KUKA KRL program: MyProgram_259().src

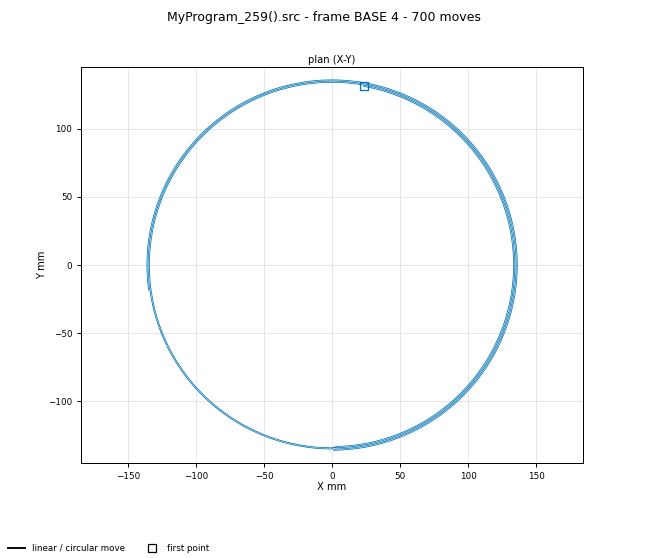
[picture p0: tool path of MyProgram_259().src in frame BASE 4, 700 of 700 moves have a stored position in this frame; points joined in program order, loops and branches not executed]
&ACCESS RVP
&REL 1
&PARAM TEMPLATE = C:\KRC\Roboter\Template\vorgabe
&PARAM EDITMASK = *
DEF MyProgram_259()
; ---- Setting reference (Base) ----
$BASE = BASE_DATA[4]

; --------------------------
; ---- Setting tool (TCP) ----
$TOOL = TOOL_DATA[3]
; --------------------------

$VEL.CP = VEL_APROX_PRINT
Startdeposition()
$VEL.CP = VEL_PRINT
LIN {X 23.111,Y 131.2816,Z 167,A 79.654,B 11.3384,C -0.0148,E1 11.3678,E2 371.0348} C_DIS
LIN {X 26.5577,Y 130.6274,Z 167,A 78.0949,B 11.3384,C -0.0129,E1 11.3721,E2 372.5994} C_DIS
LIN {X 29.5661,Y 129.9795,Z 167,A 76.8546,B 11.3384,C -0.0141,E1 11.3755,E2 373.8297} C_DIS
LIN {X 32.4376,Y 129.2932,Z 167,A 75.5169,B 11.3384,C -0.0116,E1 11.3791,E2 375.1753} C_DIS
LIN {X 34.9908,Y 128.6268,Z 167,A 73.9813,B 11.3384,C -0.0011,E1 11.3834,E2 376.758} C_DIS
LIN {X 38.5081,Y 127.6173,Z 167,A 72.9209,B 11.3384,C -0.0122,E1 11.3861,E2 377.7578} C_DIS
LIN {X 42.8444,Y 126.2288,Z 167,A 70.7155,B 11.3384,C -0.0045,E1 11.392,E2 379.9924} C_DIS
LIN {X 46.2522,Y 125.0191,Z 167,A 69.2886,B 11.3384,C -0.0061,E1 11.3957,E2 381.4041} C_DIS
LIN {X 50.6858,Y 123.2893,Z 167,A 67.2139,B 11.3384,C -0.0033,E1 11.4011,E2 383.4822} C_DIS
LIN {X 54.1145,Y 121.8215,Z 167,A 65.658,B 11.3384,C -0.0027,E1 11.4051,E2 385.0325} C_DIS
LIN {X 57.2968,Y 120.3572,Z 167,A 64.0803,B 11.3384,C 0.0009,E1 11.4091,E2 386.6187} C_DIS
LIN {X 61.2926,Y 118.3745,Z 167,A 62.2048,B 11.3384,C 0.0023,E1 11.4137,E2 388.4895} C_DIS
LIN {X 64.6789,Y 116.5587,Z 167,A 60.1894,B 11.3384,C 0.0136,E1 11.4188,E2 390.5479} C_DIS
LIN {X 68.1241,Y 114.5792,Z 167,A 58.8253,B 11.3384,C 0.0075,E1 11.422,E2 391.8717} C_DIS
LIN {X 71.9938,Y 112.1881,Z 167,A 56.8981,B 11.3384,C 0.0098,E1 11.4265,E2 393.7959} C_DIS
LIN {X 77.218,Y 108.6591,Z 167,A 54.1798,B 11.3384,C 0.0144,E1 11.4328,E2 396.5158} C_DIS
LIN {X 80.7271,Y 106.0778,Z 167,A 51.9721,B 11.3384,C 0.026,E1 11.4378,E2 398.7636} C_DIS
LIN {X 83.987,Y 103.5161,Z 167,A 50.5474,B 11.3384,C 0.0203,E1 11.4408,E2 400.1466} C_DIS
LIN {X 87.3612,Y 100.6848,Z 167,A 48.6571,B 11.3384,C 0.0237,E1 11.4448,E2 402.0372} C_DIS
LIN {X 90.7212,Y 97.6676,Z 167,A 46.7628,B 11.3384,C 0.0263,E1 11.4487,E2 403.9266} C_DIS
LIN {X 93.9495,Y 94.5662,Z 167,A 44.8876,B 11.3384,C 0.0289,E1 11.4524,E2 405.7967} C_DIS
LIN {X 97.0915,Y 91.3375,Z 167,A 42.9827,B 11.3384,C 0.0321,E1 11.4561,E2 407.6987} C_DIS
LIN {X 100.0588,Y 88.0771,Z 167,A 41.1296,B 11.3384,C 0.0351,E1 11.4596,E2 409.5477} C_DIS
LIN {X 102.7672,Y 84.9011,Z 167,A 38.5566,B 11.3384,C 0.0591,E1 11.4643,E2 412.2138} C_DIS
LIN {X 106.531,Y 80.1277,Z 167,A 36.9658,B 11.3384,C 0.0388,E1 11.4668,E2 413.6849} C_DIS
LIN {X 109.5214,Y 75.9892,Z 167,A 34.5744,B 11.3384,C 0.0491,E1 11.4707,E2 416.1011} C_DIS
LIN {X 111.9973,Y 72.291,Z 167,A 32.6754,B 11.3384,C 0.0533,E1 11.4737,E2 417.9997} C_DIS
LIN {X 113.8063,Y 69.4083,Z 167,A 30.2613,B 11.3382,C 0.0816,E1 11.4773,E2 420.5274} C_DIS
LIN {X 117.3478,Y 63.2361,Z 167,A 28.3,B 11.3383,C 0.0609,E1 11.4798,E2 422.3608} C_DIS
LIN {X 120.1649,Y 57.6993,Z 167,A 25.6079,B 11.3383,C 0.0684,E1 11.4832,E2 425.0575} C_DIS
LIN {X 121.4581,Y 54.9269,Z 167,A 24.248,B 11.3383,C 0.0731,E1 11.4847,E2 426.4238} C_DIS
LIN {X 122.6861,Y 52.1301,Z 167,A 22.924,B 11.3383,C 0.0769,E1 11.4862,E2 427.7503} C_DIS
LIN {X 124.6025,Y 47.3646,Z 167,A 20.8006,B 11.3382,C 0.0806,E1 11.4884,E2 429.8652} C_DIS
LIN {X 125.7921,Y 44.1059,Z 167,A 19.5229,B 11.3382,C 0.0791,E1 11.4896,E2 431.1185} C_DIS
LIN {X 127.1799,Y 39.931,Z 167,A 17.2589,B 11.3381,C 0.0942,E1 11.4915,E2 433.429} C_DIS
LIN {X 128.6725,Y 34.8197,Z 167,A 15.1937,B 11.3381,C 0.0947,E1 11.4931,E2 435.4693} C_DIS
LIN {X 129.5781,Y 31.2779,Z 167,A 13.6311,B 11.3381,C 0.0989,E1 11.4941,E2 437.0322} C_DIS
LIN {X 130.56,Y 26.8888,Z 167,A 11.7393,B 11.3381,C 0.1034,E1 11.4953,E2 438.9209} C_DIS
LIN {X 131.2572,Y 23.2472,Z 167,A 10.156,B 11.338,C 0.1077,E1 11.4961,E2 440.5045} C_DIS
LIN {X 131.9587,Y 18.8608,Z 167,A 8.3069,B 11.338,C 0.1116,E1 11.4968,E2 442.3481} C_DIS
LIN {X 132.4922,Y 14.6572,Z 167,A 6.5104,B 11.3379,C 0.1163,E1 11.4974,E2 444.1434} C_DIS
LIN {X 132.8356,Y 11.1164,Z 167,A 5.002,B 11.3379,C 0.1202,E1 11.4978,E2 445.6509} C_DIS
LIN {X 133.1209,Y 6.9099,Z 167,A 3.2192,B 11.3379,C 0.1247,E1 11.4981,E2 447.432} C_DIS
LIN {X 133.2576,Y 3.3765,Z 167,A 1.6311,B 11.3377,C 0.131,E1 11.4983,E2 449.0299} C_DIS
LIN {X 133.2963,Y -1.0793,Z 167,A -0.2205,B 11.3377,C 0.135,E1 11.4983,E2 450.8758} C_DIS
LIN {X 133.166,Y -6.0129,Z 167,A -2.6544,B 11.3375,C 0.1496,E1 11.498,E2 453.3496} C_DIS
LIN {X 132.9435,Y -9.7408,Z 167,A -3.8408,B 11.3375,C 0.1431,E1 11.4978,E2 454.4872} C_DIS
LIN {X 132.5722,Y -13.9132,Z 167,A -5.6427,B 11.3375,C 0.1484,E1 11.4973,E2 456.2913} C_DIS
LIN {X 132.1367,Y -17.5729,Z 167,A -7.2609,B 11.3375,C 0.154,E1 11.4967,E2 457.9154} C_DIS
LIN {X 131.5062,Y -21.7936,Z 167,A -9.0238,B 11.3375,C 0.1574,E1 11.496,E2 459.6716} C_DIS
LIN {X 130.8011,Y -25.6973,Z 167,A -10.6485,B 11.3374,C 0.1603,E1 11.4951,E2 461.2886} C_DIS
LIN {X 130.0562,Y -29.2303,Z 167,A -12.2687,B 11.3373,C 0.1666,E1 11.4942,E2 462.9187} C_DIS
LIN {X 127.6873,Y -38.2794,Z 167,A -16.8884,B 11.3368,C 0.1941,E1 11.4907,E2 467.6153} C_DIS
LIN {X 126.0223,Y -43.4421,Z 167,A -18.4516,B 11.3371,C 0.1802,E1 11.4894,E2 469.0884} C_DIS
LIN {X 124.9261,Y -46.5005,Z 167,A -20.042,B 11.3369,C 0.1893,E1 11.4878,E2 470.704} C_DIS
LIN {X 123.1296,Y -51.0683,Z 167,A -21.9539,B 11.3369,C 0.1899,E1 11.4858,E2 472.5943} C_DIS
LIN {X 121.6299,Y -54.5429,Z 167,A -23.6333,B 11.3369,C 0.1957,E1 11.4839,E2 474.2819} C_DIS
LIN {X 118.9639,Y -60.137,Z 167,A -26.2388,B 11.3367,C 0.2014,E1 11.4808,E2 476.8835} C_DIS
LIN {X 117.2059,Y -63.4995,Z 167,A -27.7083,B 11.3367,C 0.2014,E1 11.4789,E2 478.3353} C_DIS
LIN {X 115.8849,Y -65.8787,Z 167,A -29.0352,B 11.3366,C 0.2087,E1 11.477,E2 479.6826} C_DIS
LIN {X 113.6486,Y -69.6653,Z 167,A -30.9028,B 11.3366,C 0.213,E1 11.4743,E2 481.5497} C_DIS
LIN {X 111.1338,Y -73.6117,Z 167,A -32.8818,B 11.3364,C 0.2172,E1 11.4713,E2 483.5271} C_DIS
LIN {X 108.6815,Y -77.1866,Z 167,A -34.7672,B 11.3364,C 0.2224,E1 11.4683,E2 485.4173} C_DIS
LIN {X 106.0494,Y -80.7643,Z 167,A -36.6339,B 11.3363,C 0.2259,E1 11.4652,E2 487.2809} C_DIS
LIN {X 103.5315,Y -83.968,Z 167,A -38.5461,B 11.3361,C 0.2343,E1 11.4618,E2 489.2146} C_DIS
LIN {X 99.5166,Y -88.6895,Z 167,A -41.0194,B 11.3361,C 0.2354,E1 11.4573,E2 491.6677} C_DIS
LIN {X 96.4218,Y -92.044,Z 167,A -43.0399,B 11.3359,C 0.2413,E1 11.4534,E2 493.6974} C_DIS
LIN {X 93.3721,Y -95.1363,Z 167,A -44.8374,B 11.3359,C 0.2436,E1 11.4499,E2 495.4886} C_DIS
LIN {X 89.6728,Y -98.631,Z 167,A -46.9436,B 11.3359,C 0.246,E1 11.4456,E2 497.5872} C_DIS
LIN {X 86.5709,Y -101.3649,Z 167,A -49.0209,B 11.3356,C 0.2574,E1 11.4411,E2 499.7029} C_DIS
LIN {X 83.6178,Y -103.8139,Z 167,A -50.5259,B 11.3356,C 0.2569,E1 11.4379,E2 501.1921} C_DIS
LIN {X 79.3097,Y -107.1419,Z 167,A -52.6562,B 11.3356,C 0.2559,E1 11.4332,E2 503.2993} C_DIS
LIN {X 76.0282,Y -109.4943,Z 167,A -54.1959,B 11.3356,C 0.254,E1 11.4297,E2 504.8168} C_DIS
LIN {X 71.2074,Y -112.6889,Z 167,A -56.8197,B 11.3355,C 0.2618,E1 11.4236,E2 507.4599} C_DIS
LIN {X 67.5869,Y -114.8968,Z 167,A -58.6507,B 11.3355,C 0.265,E1 11.4192,E2 509.2937} C_DIS
LIN {X 63.8199,Y -117.0312,Z 167,A -60.4111,B 11.3355,C 0.2653,E1 11.4149,E2 511.0435} C_DIS
LIN {X 60.7742,Y -118.6395,Z 167,A -61.7629,B 11.3355,C 0.2642,E1 11.4116,E2 512.3809} C_DIS
LIN {X 57.705,Y -120.1622,Z 167,A -63.3149,B 11.3353,C 0.2683,E1 11.4077,E2 513.9439} C_DIS
LIN {X 54.7635,Y -121.5313,Z 167,A -64.6557,B 11.3353,C 0.2688,E1 11.4043,E2 515.2793} C_DIS
LIN {X 50.7074,Y -123.2803,Z 167,A -66.7419,B 11.3352,C 0.2759,E1 11.3988,E2 517.3901} C_DIS
LIN {X 47.1663,Y -124.6768,Z 167,A -68.2475,B 11.3352,C 0.2746,E1 11.395,E2 518.8811} C_DIS
LIN {X 44.1745,Y -125.7683,Z 167,A -70.4197,B 11.3347,C 0.2961,E1 11.389,E2 521.1519} C_DIS
LIN {X 38.5187,Y -127.6141,Z 167,A -71.8598,B 11.3353,C 0.2709,E1 11.3855,E2 522.4583} C_DIS
LIN {X 32.3264,Y -129.3214,Z 167,A -75.0203,B 11.335,C 0.2834,E1 11.3769,E2 525.6698} C_DIS
LIN {X 28.9097,Y -130.1294,Z 167,A -76.5137,B 11.335,C 0.2842,E1 11.3728,E2 527.1625} C_DIS
LIN {X 25.3413,Y -130.8692,Z 167,A -78.0214,B 11.335,C 0.2838,E1 11.3687,E2 528.6639} C_DIS
LIN {X 21.8863,Y -131.4908,Z 167,A -79.4748,B 11.335,C 0.2834,E1 11.3647,E2 530.1116} C_DIS
LIN {X 18.2129,Y -132.0513,Z 167,A -81.1212,B 11.335,C 0.2855,E1 11.3601,E2 531.7651} C_DIS
LIN {X 14.4448,Y -132.515,Z 167,A -82.6877,B 11.335,C 0.2847,E1 11.3558,E2 533.3245} C_DIS
LIN {X 11.1181,Y -132.8355,Z 167,A -84.1509,B 11.335,C 0.2859,E1 11.3517,E2 534.7917} C_DIS
LIN {X 6.9099,Y -133.1209,Z 167,A -85.9699,B 11.335,C 0.2866,E1 11.3466,E2 536.6125} C_DIS
LIN {X 3.1394,Y -133.2642,Z 167,A -87.6442,B 11.3349,C 0.2883,E1 11.3419,E2 538.294} C_DIS
LIN {X 3.1394,Y -133.2642,Z 167,A -87.6442,B 11.3349,C 0.2883,E1 11.3419,E2 538.294} C_DIS
Enddeposition()
LIN {X 0.9649,Y -134.2111,Z 167,A -88.1707,B 11.0146,C 0.3002,E1 11.0204,E2 538.9013} C_DIS
Startdeposition()
$VEL.CP = VEL_PRINT
LIN {X 3.4581,Y -134.1713,Z 167,A -86.6173,B 11.0149,C 0.2884,E1 11.0249,E2 537.2868} C_DIS
LIN {X 7.1388,Y -134.0261,Z 167,A -85.0914,B 11.0149,C 0.2891,E1 11.0291,E2 535.7658} C_DIS
LIN {X 11.0919,Y -133.7565,Z 167,A -83.3861,B 11.0149,C 0.2882,E1 11.0339,E2 534.0579} C_DIS
LIN {X 14.5172,Y -133.4281,Z 167,A -81.9055,B 11.0149,C 0.2873,E1 11.038,E2 532.575} C_DIS
LIN {X 17.6741,Y -133.0468,Z 167,A -80.5898,B 11.0149,C 0.2876,E1 11.0416,E2 531.2637} C_DIS
LIN {X 20.9035,Y -132.5781,Z 167,A -79.2392,B 11.0149,C 0.2878,E1 11.0454,E2 529.9175} C_DIS
LIN {X 23.8519,Y -132.0791,Z 167,A -77.8862,B 11.015,C 0.2852,E1 11.0491,E2 528.5541} C_DIS
LIN {X 27.4798,Y -131.374,Z 167,A -76.2645,B 11.015,C 0.283,E1 11.0536,E2 526.926} C_DIS
LIN {X 31.1737,Y -130.5451,Z 167,A -74.6858,B 11.015,C 0.2826,E1 11.0578,E2 525.3507} C_DIS
LIN {X 37.1831,Y -128.9629,Z 167,A -72.1203,B 11.015,C 0.2824,E1 11.0647,E2 522.7943} C_DIS
LIN {X 41.6665,Y -127.5844,Z 167,A -69.7848,B 11.0153,C 0.2721,E1 11.0711,E2 520.4156} C_DIS
LIN {X 44.8752,Y -126.4926,Z 167,A -68.7096,B 11.0151,C 0.2798,E1 11.0738,E2 519.3857} C_DIS
LIN {X 47.7371,Y -125.4407,Z 167,A -67.2008,B 11.0153,C 0.2731,E1 11.0778,E2 517.8501} C_DIS
LIN {X 51.3045,Y -124.0231,Z 167,A -65.8734,B 11.0152,C 0.2789,E1 11.0811,E2 516.56} C_DIS
LIN {X 53.6246,Y -123.0375,Z 167,A -64.6565,B 11.0152,C 0.274,E1 11.0843,E2 515.3247} C_DIS
LIN {X 56.6,Y -121.6971,Z 167,A -63.2535,B 11.0153,C 0.2719,E1 11.0879,E2 513.9192} C_DIS
LIN {X 60.1418,Y -119.9889,Z 167,A -61.6059,B 11.0153,C 0.2703,E1 11.092,E2 512.274} C_DIS
LIN {X 63.0439,Y -118.489,Z 167,A -60.1857,B 11.0154,C 0.2676,E1 11.0955,E2 510.8494} C_DIS
LIN {X 66.5933,Y -116.5313,Z 167,A -58.4086,B 11.0155,C 0.2637,E1 11.0999,E2 509.0649} C_DIS
LIN {X 70.5341,Y -114.1898,Z 167,A -56.2378,B 11.0157,C 0.255,E1 11.1051,E2 506.8655} C_DIS
LIN {X 73.337,Y -112.4092,Z 167,A -54.7783,B 11.0158,C 0.2515,E1 11.1085,E2 505.3993} C_DIS
LIN {X 76.4215,Y -110.336,Z 167,A -53.5539,B 11.0157,C 0.258,E1 11.1113,E2 504.2187} C_DIS
LIN {X 79.6868,Y -108.0014,Z 167,A -51.5499,B 11.0159,C 0.2474,E1 11.1159,E2 502.1767} C_DIS
LIN {X 82.426,Y -105.9255,Z 167,A -50.5266,B 11.0157,C 0.2561,E1 11.118,E2 501.2073} C_DIS
LIN {X 87.7566,Y -101.553,Z 167,A -47.6665,B 11.0157,C 0.2525,E1 11.1242,E2 498.3548} C_DIS
LIN {X 92.6598,Y -97.0998,Z 167,A -44.6294,B 11.016,C 0.2412,E1 11.1305,E2 495.2887} C_DIS
LIN {X 95.2574,Y -94.5527,Z 167,A -42.9732,B 11.0162,C 0.2352,E1 11.1337,E2 493.618} C_DIS
LIN {X 98.363,Y -91.3179,Z 167,A -40.9009,B 11.0163,C 0.2268,E1 11.1377,E2 491.5238} C_DIS
LIN {X 100.8242,Y -88.5928,Z 167,A -39.0555,B 11.0166,C 0.2158,E1 11.1412,E2 489.6418} C_DIS
LIN {X 104.2283,Y -84.5624,Z 167,A -37.4959,B 11.0163,C 0.2288,E1 11.1438,E2 488.1666} C_DIS
LIN {X 106.7196,Y -81.395,Z 167,A -35.7052,B 11.0164,C 0.2228,E1 11.1469,E2 486.3652} C_DIS
LIN {X 109.3532,Y -77.8213,Z 167,A -33.8282,B 11.0165,C 0.2187,E1 11.15,E2 484.4882} C_DIS
LIN {X 111.8562,Y -74.1793,Z 167,A -31.9264,B 11.0166,C 0.2135,E1 11.1529,E2 482.5825} C_DIS
LIN {X 114.2768,Y -70.3923,Z 167,A -30.0485,B 11.0166,C 0.2097,E1 11.1557,E2 480.7075} C_DIS
LIN {X 116.627,Y -66.4255,Z 167,A -28.3583,B 11.0166,C 0.212,E1 11.1581,E2 479.0496} C_DIS
LIN {X 118.0933,Y -63.7829,Z 167,A -26.7976,B 11.0168,C 0.2014,E1 11.1602,E2 477.4538} C_DIS
LIN {X 120.0797,Y -59.9578,Z 167,A -25.1134,B 11.0168,C 0.2006,E1 11.1623,E2 475.7869} C_DIS
LIN {X 122.5989,Y -54.6188,Z 167,A -23.0142,B 11.0168,C 0.205,E1 11.1648,E2 473.737} C_DIS
LIN {X 123.5234,Y -52.5008,Z 167,A -21.5505,B 11.017,C 0.1896,E1 11.1664,E2 472.2131} C_DIS
LIN {X 125.265,Y -48.1931,Z 167,A -19.6114,B 11.0171,C 0.1853,E1 11.1684,E2 470.2773} C_DIS
LIN {X 126.4758,Y -44.922,Z 167,A -17.9558,B 11.0172,C 0.1767,E1 11.17,E2 468.5993} C_DIS
LIN {X 127.8925,Y -40.7091,Z 167,A -16.3587,B 11.0172,C 0.1793,E1 11.1713,E2 467.0373} C_DIS
LIN {X 128.9537,Y -37.2145,Z 167,A -13.9995,B 11.0176,C 0.1534,E1 11.1732,E2 464.5766} C_DIS
LIN {X 130.4933,Y -31.3885,Z 167,A -12.4345,B 11.0173,C 0.173,E1 11.1742,E2 463.1344} C_DIS
LIN {X 131.1608,Y -28.4709,Z 167,A -11.0132,B 11.0174,C 0.1655,E1 11.1751,E2 461.6939} C_DIS
LIN {X 131.8437,Y -25.1198,Z 167,A -9.5944,B 11.0174,C 0.1624,E1 11.1758,E2 460.2785} C_DIS
LIN {X 132.4581,Y -21.6521,Z 167,A -8.115,B 11.0175,C 0.1586,E1 11.1765,E2 458.8005} C_DIS
LIN {X 132.9732,Y -18.2335,Z 167,A -6.4935,B 11.0176,C 0.1504,E1 11.1772,E2 457.1594} C_DIS
LIN {X 133.447,Y -14.3415,Z 167,A -4.9675,B 11.0176,C 0.1495,E1 11.1777,E2 455.6498} C_DIS
LIN {X 133.8003,Y -10.5737,Z 167,A -3.0213,B 11.0178,C 0.1359,E1 11.1781,E2 453.6609} C_DIS
LIN {X 134.0321,Y -7.0191,Z 167,A -2.0944,B 11.0177,C 0.1473,E1 11.1783,E2 452.8058} C_DIS
LIN {X 134.1683,Y -3.5667,Z 167,A -0.4639,B 11.0177,C 0.1388,E1 11.1784,E2 451.1547} C_DIS
LIN {X 134.2162,Y 0.2718,Z 167,A 1.2538,B 11.0179,C 0.1319,E1 11.1784,E2 449.4255} C_DIS
LIN {X 134.1522,Y 4.1432,Z 167,A 2.7921,B 11.0179,C 0.1301,E1 11.1784,E2 447.8997} C_DIS
LIN {X 133.9748,Y 8.0368,Z 167,A 4.4428,B 11.0179,C 0.1255,E1 11.1781,E2 446.249} C_DIS
LIN {X 133.745,Y 11.2285,Z 167,A 5.8177,B 11.0179,C 0.1213,E1 11.1778,E2 444.8715} C_DIS
LIN {X 133.4295,Y 14.5046,Z 167,A 7.2042,B 11.018,C 0.1177,E1 11.1774,E2 443.486} C_DIS
LIN {X 132.9148,Y 18.6428,Z 167,A 9.0024,B 11.018,C 0.1121,E1 11.1767,E2 441.6838} C_DIS
LIN {X 132.352,Y 22.2878,Z 167,A 10.5432,B 11.0181,C 0.1084,E1 11.1761,E2 440.1457} C_DIS
LIN {X 131.5324,Y 26.7015,Z 167,A 12.4115,B 11.0181,C 0.1042,E1 11.1751,E2 438.2816} C_DIS
LIN {X 130.7762,Y 30.1897,Z 167,A 13.9008,B 11.0181,C 0.1008,E1 11.1742,E2 436.7951} C_DIS
LIN {X 129.774,Y 34.2426,Z 167,A 15.687,B 11.0182,C 0.0956,E1 11.1729,E2 435.0068} C_DIS
LIN {X 128.713,Y 38.0367,Z 167,A 17.8826,B 11.0184,C 0.0773,E1 11.1712,E2 432.7464} C_DIS
LIN {X 127.2912,Y 42.5521,Z 167,A 19.3912,B 11.0184,C 0.0853,E1 11.1699,E2 431.2993} C_DIS
LIN {X 125.6178,Y 47.2642,Z 167,A 21.5575,B 11.0184,C 0.0786,E1 11.1678,E2 429.1275} C_DIS
LIN {X 124.3162,Y 50.5902,Z 167,A 22.9402,B 11.0184,C 0.0782,E1 11.1664,E2 427.761} C_DIS
LIN {X 123.0436,Y 53.6106,Z 167,A 24.3908,B 11.0184,C 0.0731,E1 11.1648,E2 426.303} C_DIS
LIN {X 121.2172,Y 57.6205,Z 167,A 26.6027,B 11.0184,C 0.0595,E1 11.1621,E2 424.0491} C_DIS
LIN {X 119.4032,Y 61.2922,Z 167,A 27.8665,B 11.0184,C 0.0677,E1 11.1606,E2 422.8436} C_DIS
LIN {X 117.7875,Y 64.3453,Z 167,A 30.052,B 11.0186,C 0.0453,E1 11.1575,E2 420.5697} C_DIS
LIN {X 115.0538,Y 69.1157,Z 167,A 31.6805,B 11.0185,C 0.0583,E1 11.1553,E2 419.0281} C_DIS
LIN {X 112.9618,Y 72.4834,Z 167,A 33.4274,B 11.0185,C 0.0527,E1 11.1527,E2 417.2735} C_DIS
LIN {X 110.5086,Y 76.1717,Z 167,A 35.5581,B 11.0185,C 0.0419,E1 11.1493,E2 415.1123} C_DIS
LIN {X 108.4311,Y 79.1016,Z 167,A 36.8459,B 11.0185,C 0.0447,E1 11.1473,E2 413.8538} C_DIS
LIN {X 104.0946,Y 84.7265,Z 167,A 39.6481,B 11.0185,C 0.0438,E1 11.1425,E2 411.078} C_DIS
LIN {X 101.8923,Y 87.3627,Z 167,A 41.2888,B 11.0185,C 0.0361,E1 11.1395,E2 409.4154} C_DIS
LIN {X 98.9133,Y 90.7214,Z 167,A 43.137,B 11.0185,C 0.0337,E1 11.136,E2 407.5747} C_DIS
LIN {X 96.0763,Y 93.7212,Z 167,A 44.944,B 11.0186,C 0.0289,E1 11.1325,E2 405.7616} C_DIS
LIN {X 92.8275,Y 96.9395,Z 167,A 46.8552,B 11.0186,C 0.026,E1 11.1287,E2 403.8546} C_DIS
LIN {X 89.4146,Y 100.0962,Z 167,A 48.8088,B 11.0186,C 0.023,E1 11.1247,E2 401.9041} C_DIS
LIN {X 85.9783,Y 103.0635,Z 167,A 50.7296,B 11.0186,C 0.0198,E1 11.1206,E2 399.9848} C_DIS
LIN {X 80.098,Y 107.6964,Z 167,A 54.5537,B 11.0186,C -0.0016,E1 11.1119,E2 396.0832} C_DIS
LIN {X 75.4981,Y 110.97,Z 167,A 56.1084,B 11.0186,C 0.016,E1 11.1086,E2 394.6322} C_DIS
LIN {X 72.82,Y 112.7455,Z 167,A 57.6162,B 11.0186,C 0.0104,E1 11.105,E2 393.1078} C_DIS
LIN {X 69.1453,Y 115.0359,Z 167,A 59.8176,B 11.0186,C -0.0011,E1 11.0997,E2 390.8633} C_DIS
LIN {X 65.8028,Y 116.9795,Z 167,A 61.1132,B 11.0186,C 0.0054,E1 11.0966,E2 389.6106} C_DIS
LIN {X 62.0142,Y 119.0297,Z 167,A 62.8825,B 11.0186,C 0.0047,E1 11.0923,E2 387.8495} C_DIS
LIN {X 59.3391,Y 120.385,Z 167,A 64.1738,B 11.0186,C 0.0028,E1 11.0891,E2 386.5568} C_DIS
LIN {X 56.0192,Y 121.9657,Z 167,A 65.6933,B 11.0186,C 0.0021,E1 11.0852,E2 385.0434} C_DIS
LIN {X 52.8538,Y 123.3708,Z 167,A 67.2391,B 11.0186,C -0.0012,E1 11.0813,E2 383.4895} C_DIS
LIN {X 48.4852,Y 125.1515,Z 167,A 69.1967,B 11.0186,C -0.0019,E1 11.0762,E2 381.5388} C_DIS
LIN {X 44.9095,Y 126.4802,Z 167,A 70.7713,B 11.0186,C -0.0021,E1 11.0721,E2 379.9709} C_DIS
LIN {X 41.0761,Y 127.7753,Z 167,A 72.4779,B 11.0186,C -0.0032,E1 11.0676,E2 378.2669} C_DIS
LIN {X 36.346,Y 129.2003,Z 167,A 74.3767,B 11.0186,C 0.0002,E1 11.0626,E2 376.3937} C_DIS
LIN {X 33.4824,Y 129.9726,Z 167,A 75.9585,B 11.0186,C -0.0082,E1 11.0582,E2 374.7742} C_DIS
LIN {X 29.8794,Y 130.8471,Z 167,A 77.4687,B 11.0186,C -0.0075,E1 11.0541,E2 373.2731} C_DIS
LIN {X 26.6862,Y 131.5355,Z 167,A 78.8545,B 11.0186,C -0.008,E1 11.0503,E2 371.8887} C_DIS
LIN {X 23.5582,Y 132.1316,Z 167,A 80.2365,B 11.0186,C -0.0092,E1 11.0465,E2 370.5043} C_DIS
LIN {X 19.7626,Y 132.7547,Z 167,A 81.8258,B 11.0186,C -0.0086,E1 11.0421,E2 368.9219} C_DIS
LIN {X 16.2843,Y 133.2244,Z 167,A 83.4219,B 11.0186,C -0.0114,E1 11.0377,E2 367.3145} C_DIS
LIN {X 12.6554,Y 133.6176,Z 167,A 84.9258,B 11.0186,C -0.0105,E1 11.0335,E2 365.8177} C_DIS
LIN {X 8.378,Y 133.9538,Z 167,A 86.7607,B 11.0186,C -0.0109,E1 11.0284,E2 363.9831} C_DIS
LIN {X 4.659,Y 134.1359,Z 167,A 88.3908,B 11.0186,C -0.0119,E1 11.0239,E2 362.3488} C_DIS
LIN {X 0.7067,Y 134.2137,Z 167,A 90.0012,B 11.0186,C -0.0102,E1 11.0194,E2 360.7485} C_DIS
LIN {X -3.1537,Y 134.1797,Z 167,A 91.7456,B 11.0186,C -0.0122,E1 11.0145,E2 358.9933} C_DIS
LIN {X -7.024,Y 134.0319,Z 167,A 93.4354,B 11.0186,C -0.0127,E1 11.0098,E2 357.2999} C_DIS
LIN {X -11.2551,Y 133.7427,Z 167,A 95.1269,B 11.0186,C -0.0095,E1 11.0051,E2 355.6237} C_DIS
LIN {X -14.8408,Y 133.3933,Z 167,A 96.6516,B 11.0186,C -0.0087,E1 11.0009,E2 354.1015} C_DIS
LIN {X -18.5922,Y 132.922,Z 167,A 98.3458,B 11.0186,C -0.0098,E1 10.9962,E2 352.3986} C_DIS
LIN {X -22.3311,Y 132.3448,Z 167,A 99.9063,B 11.0186,C -0.0077,E1 10.9919,E2 350.8456} C_DIS
LIN {X -26.2813,Y 131.6179,Z 167,A 102.4045,B 11.0186,C -0.0243,E1 10.9848,E2 348.254} C_DIS
LIN {X -31.9508,Y 130.3577,Z 167,A 103.8647,B 11.0186,C 0.0003,E1 10.9812,E2 346.9183} C_DIS
LIN {X -37.324,Y 128.9217,Z 167,A 107.0422,B 11.0186,C -0.0156,E1 10.9723,E2 343.6461} C_DIS
LIN {X -41.7584,Y 127.5555,Z 167,A 108.6732,B 11.0186,C -0.0059,E1 10.9681,E2 342.0589} C_DIS
LIN {X -45.7248,Y 126.1863,Z 167,A 110.2459,B 11.0186,C 0.0007,E1 10.9641,E2 340.5137} C_DIS
LIN {X -48.5561,Y 125.1239,Z 167,A 111.5711,B 11.0186,C 0.0014,E1 10.9606,E2 339.1854} C_DIS
LIN {X -51.5415,Y 123.9241,Z 167,A 113.1191,B 11.0186,C -0.0008,E1 10.9565,E2 337.6176} C_DIS
LIN {X -55.4809,Y 122.2133,Z 167,A 114.8021,B 11.0186,C 0.0047,E1 10.9523,E2 335.9543} C_DIS
LIN {X -58.4461,Y 120.8228,Z 167,A 116.1979,B 11.0186,C 0.0066,E1 10.9488,E2 334.5599} C_DIS
LIN {X -61.3975,Y 119.3496,Z 167,A 118.422,B 11.0186,C -0.0091,E1 10.943,E2 332.2386} C_DIS
LIN {X -66.5655,Y 116.5471,Z 167,A 120.2297,B 11.0186,C 0.0098,E1 10.9388,E2 330.5181} C_DIS
LIN {X -70.4643,Y 114.2326,Z 167,A 122.2382,B 11.0186,C 0.0113,E1 10.934,E2 328.5027} C_DIS
LIN {X -74.2093,Y 111.8361,Z 167,A 124.1252,B 11.0186,C 0.0146,E1 10.9296,E2 326.6187} C_DIS
LIN {X -77.8481,Y 109.3341,Z 167,A 126.0044,B 11.0186,C 0.018,E1 10.9253,E2 324.7421} C_DIS
LIN {X -81.3265,Y 106.772,Z 167,A 127.8942,B 11.0186,C 0.0204,E1 10.9211,E2 322.8487} C_DIS
LIN {X -84.8121,Y 104.0247,Z 167,A 129.7646,B 11.0186,C 0.0245,E1 10.917,E2 320.9831} C_DIS
LIN {X -88.0058,Y 101.3374,Z 167,A 131.5737,B 11.0186,C 0.0274,E1 10.9132,E2 319.1726} C_DIS
LIN {X -91.1488,Y 98.5204,Z 167,A 133.4375,B 11.0186,C 0.0297,E1 10.9093,E2 317.3031} C_DIS
LIN {X -94.371,Y 95.438,Z 167,A 135.3216,B 11.0186,C 0.0341,E1 10.9056,E2 315.4234} C_DIS
LIN {X -97.345,Y 92.403,Z 167,A 137.1687,B 11.0186,C 0.0373,E1 10.902,E2 313.5742} C_DIS
LIN {X -100.2699,Y 89.2207,Z 167,A 139.065,B 11.0186,C 0.0404,E1 10.8984,E2 311.6738} C_DIS
LIN {X -103.2211,Y 85.7885,Z 167,A 140.9602,B 11.0186,C 0.0455,E1 10.895,E2 309.7851} C_DIS
LIN {X -105.8942,Y 82.4664,Z 167,A 142.8217,B 11.0186,C 0.049,E1 10.8918,E2 307.9207} C_DIS
LIN {X -108.4559,Y 79.0674,Z 167,A 144.6843,B 11.0186,C 0.0524,E1 10.8887,E2 306.0546} C_DIS
LIN {X -111.0514,Y 75.3778,Z 167,A 146.6154,B 11.0186,C 0.057,E1 10.8856,E2 304.125} C_DIS
LIN {X -114.9038,Y 69.3637,Z 167,A 149.5451,B 11.0184,C 0.0671,E1 10.8813,E2 301.2131} C_DIS
LIN {X -117.0802,Y 65.6235,Z 167,A 151.5505,B 11.0184,C 0.0687,E1 10.8785,E2 299.1908} C_DIS
LIN {X -118.9929,Y 62.0844,Z 167,A 153.2308,B 11.0184,C 0.0739,E1 10.8763,E2 297.5168} C_DIS
LIN {X -120.9316,Y 58.2183,Z 167,A 154.8959,B 11.0184,C 0.0825,E1 10.8743,E2 295.8756} C_DIS
LIN {X -122.2291,Y 55.4457,Z 167,A 156.6317,B 11.0184,C 0.0774,E1 10.8722,E2 294.0896} C_DIS
LIN {X -123.9786,Y 51.4112,Z 167,A 158.2839,B 11.0184,C 0.087,E1 10.8704,E2 292.4666} C_DIS
LIN {X -125.1515,Y 48.4852,Z 167,A 159.6768,B 11.0183,C 0.0898,E1 10.869,E2 291.0695} C_DIS
LIN {X -126.3765,Y 45.1971,Z 167,A 161.2075,B 11.0183,C 0.0933,E1 10.8675,E2 289.5367} C_DIS
LIN {X -127.4498,Y 42.0758,Z 167,A 162.6158,B 11.0183,C 0.0973,E1 10.8663,E2 288.13} C_DIS
LIN {X -128.4081,Y 39.0529,Z 167,A 163.9677,B 11.0182,C 0.1011,E1 10.8652,E2 286.7799} C_DIS
LIN {X -129.4526,Y 35.4439,Z 167,A 165.8858,B 11.0182,C 0.0994,E1 10.8637,E2 284.8256} C_DIS
LIN {X -130.6762,Y 30.6274,Z 167,A 167.7329,B 11.0181,C 0.111,E1 10.8625,E2 283.0141} C_DIS
LIN {X -131.3468,Y 27.6096,Z 167,A 169.0639,B 11.0181,C 0.1146,E1 10.8617,E2 281.6831} C_DIS
LIN {X -132.0375,Y 24.084,Z 167,A 171.376,B 11.0181,C 0.1033,E1 10.8605,E2 279.2781} C_DIS
LIN {X -132.9101,Y 18.6757,Z 167,A 173.0216,B 11.018,C 0.1241,E1 10.8599,E2 277.7194} C_DIS
LIN {X -133.3719,Y 15.0396,Z 167,A 174.7216,B 11.018,C 0.126,E1 10.8593,E2 276.0048} C_DIS
LIN {X -133.7558,Y 11.0997,Z 167,A 176.3237,B 11.0179,C 0.1327,E1 10.8589,E2 274.4151} C_DIS
LIN {X -134.0065,Y 7.5223,Z 167,A 177.9145,B 11.0179,C 0.136,E1 10.8586,E2 272.8187} C_DIS
LIN {X -134.1621,Y 3.7883,Z 167,A 179.4595,B 11.0177,C 0.1417,E1 10.8585,E2 271.2814} C_DIS
LIN {X -134.2176,Y 0.0186,Z 167,A -178.7535,B 11.0177,C 0.1429,E1 10.8585,E2 269.4747} C_DIS
LIN {X -134.1468,Y -4.3373,Z 167,A -177.0174,B 11.0177,C 0.1508,E1 10.8585,E2 267.7553} C_DIS
LIN {X -133.9681,Y -8.1464,Z 167,A -175.3238,B 11.0176,C 0.1542,E1 10.8588,E2 266.0555} C_DIS
LIN {X -133.6806,Y -11.991,Z 167,A -173.5768,B 11.0176,C 0.157,E1 10.8592,E2 264.2979} C_DIS
LIN {X -133.2665,Y -15.9316,Z 167,A -171.9816,B 11.0174,C 0.1639,E1 10.8597,E2 262.7159} C_DIS
LIN {X -132.827,Y -19.2568,Z 167,A -170.4903,B 11.0174,C 0.1668,E1 10.8603,E2 261.2188} C_DIS
LIN {X -131.5995,Y -26.3717,Z 167,A -167.5625,B 11.0172,C 0.1788,E1 10.8617,E2 258.3127} C_DIS
LIN {X -130.7269,Y -30.4056,Z 167,A -165.3003,B 11.0172,C 0.1737,E1 10.8631,E2 255.9912} C_DIS
LIN {X -129.9521,Y -33.5621,Z 167,A -164.0616,B 11.0172,C 0.1806,E1 10.864,E2 254.7719} C_DIS
LIN {X -128.6789,Y -38.1532,Z 167,A -162.1451,B 11.0171,C 0.1887,E1 10.8654,E2 252.8715} C_DIS
LIN {X -127.8939,Y -40.7048,Z 167,A -160.919,B 11.0171,C 0.1901,E1 10.8665,E2 251.6357} C_DIS
LIN {X -126.7072,Y -44.2614,Z 167,A -159.3669,B 11.0169,C 0.1955,E1 10.8679,E2 250.091} C_DIS
LIN {X -125.4624,Y -47.679,Z 167,A -157.8107,B 11.0169,C 0.1996,E1 10.8694,E2 248.5356} C_DIS
LIN {X -124.1252,Y -51.06,Z 167,A -156.097,B 11.0169,C 0.2005,E1 10.8712,E2 246.8034} C_DIS
LIN {X -122.249,Y -55.4012,Z 167,A -153.7844,B 11.0169,C 0.1997,E1 10.8739,E2 244.4563} C_DIS
LIN {X -120.6814,Y -58.737,Z 167,A -152.5723,B 11.0166,C 0.2113,E1 10.8753,E2 243.2897} C_DIS
LIN {X -119.4536,Y -61.1933,Z 167,A -151.3481,B 11.0166,C 0.2132,E1 10.8768,E2 242.0598} C_DIS
LIN {X -117.5946,Y -64.6975,Z 167,A -149.6442,B 11.0166,C 0.2173,E1 10.8791,E2 240.3559} C_DIS
LIN {X -115.53,Y -68.3167,Z 167,A -147.8011,B 11.0165,C 0.2204,E1 10.8817,E2 238.5061} C_DIS
LIN {X -113.439,Y -71.7343,Z 167,A -145.9335,B 11.0165,C 0.2213,E1 10.8845,E2 236.6202} C_DIS
LIN {X -110.2371,Y -76.5636,Z 167,A -143.6829,B 11.0162,C 0.2318,E1 10.888,E2 234.3985} C_DIS
LIN {X -107.9898,Y -79.7025,Z 167,A -141.844,B 11.0162,C 0.2316,E1 10.891,E2 232.5372} C_DIS
LIN {X -105.2058,Y -83.3429,Z 167,A -139.9184,B 11.0162,C 0.2367,E1 10.8943,E2 230.6164} C_DIS
LIN {X -102.481,Y -86.6716,Z 167,A -138.0112,B 11.0161,C 0.2392,E1 10.8977,E2 228.7013} C_DIS
LIN {X -99.5379,Y -90.0358,Z 167,A -136.1077,B 11.016,C 0.2433,E1 10.9013,E2 226.7992} C_DIS
LIN {X -96.3947,Y -93.393,Z 167,A -134.1691,B 11.0159,C 0.2478,E1 10.905,E2 224.8645} C_DIS
LIN {X -93.2697,Y -96.5141,Z 167,A -132.2526,B 11.0159,C 0.2509,E1 10.9088,E2 222.945} C_DIS
LIN {X -90.1678,Y -99.4181,Z 167,A -130.4028,B 11.0158,C 0.2536,E1 10.9126,E2 221.0913} C_DIS
LIN {X -86.203,Y -102.8749,Z 167,A -128.0313,B 11.0158,C 0.2549,E1 10.9177,E2 218.705} C_DIS
LIN {X -82.3143,Y -106.0121,Z 167,A -126.0006,B 11.0156,C 0.2608,E1 10.9221,E2 216.6875} C_DIS
LIN {X -78.7315,Y -108.6994,Z 167,A -124.0772,B 11.0156,C 0.2637,E1 10.9264,E2 214.7631} C_DIS
LIN {X -75.2136,Y -111.1626,Z 167,A -122.2304,B 11.0155,C 0.2663,E1 10.9307,E2 212.915} C_DIS
LIN {X -71.7133,Y -113.4522,Z 167,A -120.3394,B 11.0155,C 0.2666,E1 10.9352,E2 211.0113} C_DIS
LIN {X -67.3094,Y -116.1191,Z 167,A -118.2504,B 11.0153,C 0.2721,E1 10.9402,E2 208.936} C_DIS
LIN {X -63.196,Y -118.4086,Z 167,A -116.2878,B 11.0153,C 0.2758,E1 10.945,E2 206.9794} C_DIS
LIN {X -60.5656,Y -119.7731,Z 167,A -115.019,B 11.0153,C 0.2772,E1 10.9481,E2 205.7102} C_DIS
LIN {X -57.4549,Y -121.2963,Z 167,A -113.5441,B 11.0152,C 0.279,E1 10.9518,E2 204.2358} C_DIS
LIN {X -54.4803,Y -122.6609,Z 167,A -112.0839,B 11.0152,C 0.2791,E1 10.9556,E2 202.7677} C_DIS
LIN {X -51.5631,Y -123.9151,Z 167,A -110.7318,B 11.0152,C 0.2806,E1 10.959,E2 201.416} C_DIS
LIN {X -48.0419,Y -125.3238,Z 167,A -109.1483,B 11.0151,C 0.2829,E1 10.9631,E2 199.8368} C_DIS
LIN {X -44.1036,Y -126.7619,Z 167,A -107.3839,B 11.0151,C 0.2851,E1 10.9678,E2 198.0753} C_DIS
LIN {X -39.592,Y -128.2431,Z 167,A -105.4999,B 11.0149,C 0.2899,E1 10.9727,E2 196.2089} C_DIS
LIN {X -35.9566,Y -129.3092,Z 167,A -103.7076,B 11.0149,C 0.287,E1 10.9776,E2 194.3946} C_DIS
LIN {X -32.561,Y -130.2065,Z 167,A -102.0602,B 11.015,C 0.2845,E1 10.9821,E2 192.7285} C_DIS
LIN {X -28.5349,Y -131.147,Z 167,A -100.3541,B 11.015,C 0.2868,E1 10.9867,E2 191.0293} C_DIS
LIN {X -24.6253,Y -131.9382,Z 167,A -98.5764,B 11.015,C 0.2858,E1 10.9916,E2 189.2419} C_DIS
LIN {X -20.5521,Y -132.6325,Z 167,A -96.8925,B 11.015,C 0.2883,E1 10.9963,E2 187.5673} C_DIS
LIN {X -17.0631,Y -133.1269,Z 167,A -95.3291,B 11.015,C 0.2873,E1 11.0006,E2 185.9961} C_DIS
LIN {X -13.0127,Y -133.5833,Z 167,A -93.6553,B 11.015,C 0.2891,E1 11.0052,E2 184.3299} C_DIS
LIN {X -9.6617,Y -133.8673,Z 167,A -92.2352,B 11.0149,C 0.2896,E1 11.0092,E2 182.9111} C_DIS
LIN {X -6.3112,Y -134.0677,Z 167,A -90.6848,B 11.0149,C 0.2869,E1 11.0135,E2 181.3455} C_DIS
LIN {X -2.048,Y -134.2001,Z 167,A -88.9956,B 11.0149,C 0.2899,E1 11.0182,E2 179.6719} C_DIS
LIN {X 0.9649,Y -134.2111,Z 167,A -88.1687,B 11.0146,C 0.3006,E1 11.0204,E2 178.9012} C_DIS
Enddeposition()
LIN {X 0.9649,Y -134.2111,Z 167,A -88.1687,B 11.0146,C 0.3006,E1 11.0204,E2 178.9012} C_DIS
Startdeposition()
$VEL.CP = VEL_PRINT
LIN {X -0.0193,Y -135.1331,Z 167,A -88.8426,B 10.9264,C 0.3172,E1 10.9305,E2 179.6684} C_DIS
LIN {X -4.0821,Y -135.0699,Z 167,A -90.5664,B 10.9264,C 0.3173,E1 10.9257,E2 181.393} C_DIS
LIN {X -7.9876,Y -134.8952,Z 167,A -91.9617,B 10.9265,C 0.3112,E1 10.9219,E2 182.7564} C_DIS
LIN {X -10.4926,Y -134.7247,Z 167,A -93.286,B 10.9264,C 0.3171,E1 10.9181,E2 184.1134} C_DIS
LIN {X -14.8728,Y -134.3107,Z 167,A -95.1453,B 10.9264,C 0.3167,E1 10.9129,E2 185.9726} C_DIS
LIN {X -18.9857,Y -133.7906,Z 167,A -96.7766,B 10.9264,C 0.3133,E1 10.9085,E2 187.5888} C_DIS
LIN {X -21.8409,Y -133.3548,Z 167,A -97.8802,B 10.9266,C 0.3101,E1 10.9054,E2 188.6778} C_DIS
LIN {X -24.4062,Y -132.91,Z 167,A -99.2581,B 10.9264,C 0.316,E1 10.9016,E2 190.09} C_DIS
LIN {X -28.3606,Y -132.1213,Z 167,A -100.8138,B 10.9265,C 0.3116,E1 10.8974,E2 191.6271} C_DIS
LIN {X -31.533,Y -131.4002,Z 167,A -102.1985,B 10.9265,C 0.311,E1 10.8936,E2 193.0127} C_DIS
LIN {X -34.489,Y -130.6558,Z 167,A -103.3958,B 10.9266,C 0.3081,E1 10.8904,E2 194.1984} C_DIS
LIN {X -37.0529,Y -129.9533,Z 167,A -104.7401,B 10.9266,C 0.3122,E1 10.8867,E2 195.5699} C_DIS
LIN {X -40.9198,Y -128.7864,Z 167,A -106.4542,B 10.9266,C 0.311,E1 10.8821,E2 197.2844} C_DIS
LIN {X -45.2603,Y -127.327,Z 167,A -108.2366,B 10.9266,C 0.3058,E1 10.8775,E2 199.0474} C_DIS
LIN {X -48.6628,Y -126.0647,Z 167,A -109.8819,B 10.9266,C 0.3068,E1 10.8731,E2 200.7059} C_DIS
LIN {X -51.9079,Y -124.7633,Z 167,A -111.2464,B 10.9268,C 0.3027,E1 10.8696,E2 202.0559} C_DIS
LIN {X -54.9087,Y -123.4722,Z 167,A -112.7067,B 10.9268,C 0.3029,E1 10.8659,E2 203.5256} C_DIS
LIN {X -57.9361,Y -122.0811,Z 167,A -114.0169,B 10.9268,C 0.299,E1 10.8626,E2 204.8231} C_DIS
LIN {X -60.8608,Y -120.6502,Z 167,A -115.4098,B 10.9269,C 0.2977,E1 10.8591,E2 206.2176} C_DIS
LIN {X -63.7479,Y -119.1515,Z 167,A -116.7195,B 10.9269,C 0.2944,E1 10.8559,E2 207.5187} C_DIS
LIN {X -67.0435,Y -117.3285,Z 167,A -119.3407,B 10.9264,C 0.3146,E1 10.8492,E2 210.2652} C_DIS
LIN {X -72.1174,Y -114.2799,Z 167,A -121.1601,B 10.927,C 0.2961,E1 10.8451,E2 212} C_DIS
LIN {X -75.9366,Y -111.7787,Z 167,A -123.1234,B 10.927,C 0.2937,E1 10.8405,E2 213.9664} C_DIS
LIN {X -79.5051,Y -109.2694,Z 167,A -124.8029,B 10.9272,C 0.2871,E1 10.8368,E2 215.6246} C_DIS
LIN {X -83.077,Y -106.5793,Z 167,A -127.7538,B 10.9267,C 0.3063,E1 10.83,E2 218.7036} C_DIS
LIN {X -88.2892,Y -102.3026,Z 167,A -129.7481,B 10.9273,C 0.2829,E1 10.826,E2 220.5919} C_DIS
LIN {X -91.6912,Y -99.2654,Z 167,A -131.6721,B 10.9273,C 0.279,E1 10.822,E2 222.5141} C_DIS
LIN {X -94.8253,Y -96.2759,Z 167,A -133.5468,B 10.9275,C 0.2763,E1 10.8182,E2 224.3928} C_DIS
LIN {X -97.8539,Y -93.1959,Z 167,A -135.4214,B 10.9275,C 0.2734,E1 10.8145,E2 226.2719} C_DIS
LIN {X -100.8928,Y -89.8975,Z 167,A -137.3512,B 10.9276,C 0.2701,E1 10.8109,E2 228.2044} C_DIS
LIN {X -103.8465,Y -86.4688,Z 167,A -139.3059,B 10.9277,C 0.2666,E1 10.8074,E2 230.1624} C_DIS
LIN {X -106.6105,Y -83.0368,Z 167,A -141.1688,B 10.9278,C 0.2624,E1 10.8042,E2 232.0238} C_DIS
LIN {X -109.8746,Y -78.6663,Z 167,A -143.2225,B 10.9281,C 0.2517,E1 10.8008,E2 234.0444} C_DIS
LIN {X -114.1143,Y -72.3797,Z 167,A -146.7918,B 10.9281,C 0.2514,E1 10.7952,E2 237.6553} C_DIS
LIN {X -116.308,Y -68.7998,Z 167,A -148.552,B 10.9281,C 0.2466,E1 10.7927,E2 239.412} C_DIS
LIN {X -118.377,Y -65.1751,Z 167,A -150.4859,B 10.9281,C 0.2455,E1 10.79,E2 241.3646} C_DIS
LIN {X -120.7804,Y -60.6045,Z 167,A -153.1572,B 10.9281,C 0.2496,E1 10.7866,E2 244.0926} C_DIS
LIN {X -123.0556,Y -55.8401,Z 167,A -154.8336,B 10.9285,C 0.2324,E1 10.7847,E2 245.6994} C_DIS
LIN {X -124.591,Y -52.3204,Z 167,A -156.3677,B 10.9286,C 0.2262,E1 10.783,E2 247.2208} C_DIS
LIN {X -125.7452,Y -49.4849,Z 167,A -157.5905,B 10.9287,C 0.2212,E1 10.7818,E2 248.4335} C_DIS
LIN {X -127.0481,Y -46.0338,Z 167,A -159.2503,B 10.9287,C 0.2189,E1 10.7801,E2 250.1036} C_DIS
LIN {X -128.1288,Y -42.9346,Z 167,A -160.669,B 10.9288,C 0.2156,E1 10.7788,E2 251.5245} C_DIS
LIN {X -129.0282,Y -40.1551,Z 167,A -162.3701,B 10.9287,C 0.2214,E1 10.7774,E2 253.2806} C_DIS
LIN {X -130.1021,Y -36.5209,Z 167,A -163.3915,B 10.929,C 0.2052,E1 10.7767,E2 254.2297} C_DIS
LIN {X -131.4038,Y -31.5182,Z 167,A -165.8497,B 10.929,C 0.2044,E1 10.7749,E2 256.7184} C_DIS
LIN {X -132.3226,Y -27.4101,Z 167,A -167.5766,B 10.9291,C 0.1982,E1 10.7739,E2 258.4367} C_DIS
LIN {X -132.8505,Y -24.7293,Z 167,A -168.9493,B 10.9291,C 0.1991,E1 10.7732,E2 259.8343} C_DIS
LIN {X -133.5245,Y -20.7748,Z 167,A -170.5361,B 10.9292,C 0.1919,E1 10.7725,E2 261.4056} C_DIS
LIN {X -134.078,Y -16.8517,Z 167,A -172.3515,B 10.9292,C 0.1898,E1 10.7718,E2 263.2359} C_DIS
LIN {X -134.5201,Y -12.8351,Z 167,A -173.9693,B 10.9294,C 0.1829,E1 10.7714,E2 264.8404} C_DIS
LIN {X -134.8564,Y -8.6174,Z 167,A -175.8058,B 10.9294,C 0.1785,E1 10.771,E2 266.6803} C_DIS
LIN {X -135.0259,Y -5.3309,Z 167,A -177.0869,B 10.9296,C 0.1721,E1 10.7708,E2 267.9462} C_DIS
LIN {X -135.1061,Y -2.6282,Z 167,A -178.2995,B 10.9296,C 0.1701,E1 10.7708,E2 269.1657} C_DIS
LIN {X -135.1283,Y 0.918,Z 167,A -179.9285,B 10.9296,C 0.1682,E1 10.7708,E2 270.8082} C_DIS
LIN {X -135.0304,Y 5.2155,Z 167,A 178.3007,B 10.9297,C 0.1618,E1 10.7708,E2 272.5708} C_DIS
LIN {X -134.8516,Y 8.6956,Z 167,A 176.6893,B 10.9297,C 0.1601,E1 10.7711,E2 274.1968} C_DIS
LIN {X -134.5605,Y 12.4139,Z 167,A 175.1046,B 10.9298,C 0.1555,E1 10.7715,E2 275.7803} C_DIS
LIN {X -134.2296,Y 15.5874,Z 167,A 173.7295,B 10.9298,C 0.152,E1 10.7719,E2 277.1567} C_DIS
LIN {X -133.7589,Y 19.2073,Z 167,A 172.4381,B 10.93,C 0.1424,E1 10.7724,E2 278.4154} C_DIS
LIN {X -133.1892,Y 22.8335,Z 167,A 170.5229,B 10.93,C 0.145,E1 10.7733,E2 280.3722} C_DIS
LIN {X -132.4078,Y 26.9909,Z 167,A 168.8578,B 10.93,C 0.1373,E1 10.7742,E2 282.0199} C_DIS
LIN {X -131.5498,Y 30.9125,Z 167,A 167.1463,B 10.9301,C 0.1326,E1 10.7752,E2 283.7307} C_DIS
LIN {X -130.8496,Y 33.7489,Z 167,A 165.8734,B 10.9301,C 0.1297,E1 10.7761,E2 285.0063} C_DIS
LIN {X -129.8073,Y 37.5575,Z 167,A 164.149,B 10.9301,C 0.1259,E1 10.7774,E2 286.7349} C_DIS
LIN {X -128.8374,Y 40.76,Z 167,A 162.7852,B 10.9303,C 0.1208,E1 10.7785,E2 288.0904} C_DIS
LIN {X -127.9334,Y 43.5195,Z 167,A 161.506,B 10.9303,C 0.1183,E1 10.7796,E2 289.3741} C_DIS
LIN {X -126.6774,Y 47.0455,Z 167,A 159.8256,B 10.9303,C 0.1158,E1 10.7813,E2 291.0639} C_DIS
LIN {X -125.546,Y 49.9883,Z 167,A 158.5081,B 10.9303,C 0.1117,E1 10.7826,E2 292.3776} C_DIS
LIN {X -124.3641,Y 52.8633,Z 167,A 156.9605,B 10.9303,C 0.1127,E1 10.7843,E2 293.9513} C_DIS
LIN {X -122.8816,Y 56.2199,Z 167,A 155.7222,B 10.9304,C 0.1021,E1 10.7857,E2 295.1497} C_DIS
LIN {X -121.2868,Y 59.5803,Z 167,A 153.5846,B 10.9304,C 0.1091,E1 10.7884,E2 297.3525} C_DIS
LIN {X -119.5105,Y 63.0681,Z 167,A 152.4855,B 10.9305,C 0.0935,E1 10.7897,E2 298.3827} C_DIS
LIN {X -116.5586,Y 68.3733,Z 167,A 149.5242,B 10.9305,C 0.0947,E1 10.7938,E2 301.3877} C_DIS
LIN {X -113.2439,Y 73.7338,Z 167,A 146.9296,B 10.9305,C 0.0864,E1 10.7977,E2 303.97} C_DIS
LIN {X -110.7576,Y 77.4186,Z 167,A 145.0068,B 10.9306,C 0.0825,E1 10.8007,E2 305.8953} C_DIS
LIN {X -108.1976,Y 80.958,Z 167,A 143.1375,B 10.9306,C 0.0784,E1 10.8038,E2 307.7646} C_DIS
LIN {X -105.6859,Y 84.2099,Z 167,A 141.4164,B 10.9306,C 0.0739,E1 10.8068,E2 309.4813} C_DIS
LIN {X -103.0161,Y 87.4556,Z 167,A 139.6024,B 10.9306,C 0.0705,E1 10.81,E2 311.2972} C_DIS
LIN {X -100.1836,Y 90.6867,Z 167,A 137.7252,B 10.9307,C 0.0675,E1 10.8135,E2 313.179} C_DIS
LIN {X -97.0301,Y 94.053,Z 167,A 135.7874,B 10.9307,C 0.0629,E1 10.8172,E2 315.1125} C_DIS
LIN {X -94.0217,Y 97.0604,Z 167,A 133.9624,B 10.9307,C 0.0596,E1 10.8208,E2 316.9383} C_DIS
LIN {X -90.8283,Y 100.0551,Z 167,A 132.0637,B 10.9307,C 0.0567,E1 10.8248,E2 318.8401} C_DIS
LIN {X -87.4307,Y 103.0373,Z 167,A 130.117,B 10.9307,C 0.0535,E1 10.8289,E2 320.7884} C_DIS
LIN {X -84.0529,Y 105.8108,Z 167,A 128.3033,B 10.9308,C 0.0492,E1 10.8328,E2 322.5956} C_DIS
LIN {X -80.6043,Y 108.4609,Z 167,A 126.3957,B 10.9308,C 0.0472,E1 10.8371,E2 324.5089} C_DIS
LIN {X -76.8939,Y 111.1227,Z 167,A 124.4311,B 10.9308,C 0.0444,E1 10.8415,E2 326.4751} C_DIS
LIN {X -73.153,Y 113.6203,Z 167,A 122.5096,B 10.9308,C 0.0416,E1 10.846,E2 328.3964} C_DIS
LIN {X -69.6719,Y 115.7874,Z 167,A 120.7915,B 10.9308,C 0.0384,E1 10.8501,E2 330.1105} C_DIS
LIN {X -65.5781,Y 118.1539,Z 167,A 118.5947,B 10.9308,C 0.0394,E1 10.8555,E2 332.3283} C_DIS
LIN {X -61.4539,Y 120.3483,Z 167,A 117.0068,B 10.9308,C 0.0283,E1 10.8593,E2 333.8675} C_DIS
LIN {X -58.5503,Y 121.7877,Z 167,A 115.4733,B 10.9308,C 0.0299,E1 10.8632,E2 335.4189} C_DIS
LIN {X -55.8782,Y 123.0386,Z 167,A 114.2448,B 10.9308,C 0.0278,E1 10.8663,E2 336.6438} C_DIS
LIN {X -53.0177,Y 124.2974,Z 167,A 112.6817,B 10.9308,C 0.0313,E1 10.8704,E2 338.2341} C_DIS
LIN {X -49.1981,Y 125.8567,Z 167,A 111.112,B 10.9308,C 0.0255,E1 10.8744,E2 339.781} C_DIS
LIN {X -46.3284,Y 126.9419,Z 167,A 109.9388,B 10.9308,C 0.0213,E1 10.8774,E2 340.9379} C_DIS
LIN {X -41.5971,Y 128.57,Z 167,A 107.8175,B 10.9308,C 0.0192,E1 10.883,E2 343.0576} C_DIS
LIN {X -35.0959,Y 130.494,Z 167,A 104.7469,B 10.9308,C 0.021,E1 10.8913,E2 346.1496} C_DIS
LIN {X -31.1683,Y 131.4882,Z 167,A 102.9845,B 10.9308,C 0.0207,E1 10.8961,E2 347.9162} C_DIS
LIN {X -26.3087,Y 132.5467,Z 167,A 100.8801,B 10.9308,C 0.0193,E1 10.9019,E2 350.0187} C_DIS
LIN {X -22.6845,Y 133.214,Z 167,A 99.45,B 10.9309,C 0.0155,E1 10.9057,E2 351.4319} C_DIS
LIN {X -19.9737,Y 133.6485,Z 167,A 98.0765,B 10.9309,C 0.0196,E1 10.9096,E2 352.8298} C_DIS
LIN {X -15.5578,Y 134.2332,Z 167,A 96.2298,B 10.9309,C 0.0178,E1 10.9147,E2 354.6703} C_DIS
LIN {X -11.4227,Y 134.6474,Z 167,A 94.6395,B 10.9309,C 0.0134,E1 10.9191,E2 356.2391} C_DIS
LIN {X -8.663,Y 134.8536,Z 167,A 93.5449,B 10.9309,C 0.0114,E1 10.9221,E2 357.3237} C_DIS
LIN {X -5.2765,Y 135.028,Z 167,A 91.8561,B 10.9309,C 0.0168,E1 10.9269,E2 359.0417} C_DIS
LIN {X -0.8878,Y 135.1283,Z 167,A 90.0987,B 10.9309,C 0.0142,E1 10.9318,E2 360.7859} C_DIS
LIN {X 2.7292,Y 135.1044,Z 167,A 88.4607,B 10.9309,C 0.0166,E1 10.9364,E2 362.4357} C_DIS
LIN {X 6.1533,Y 134.9924,Z 167,A 86.9883,B 10.9309,C 0.0172,E1 10.9405,E2 363.9099} C_DIS
LIN {X 10.6051,Y 134.7164,Z 167,A 85.0968,B 10.9309,C 0.0175,E1 10.9457,E2 365.8007} C_DIS
LIN {X 14.3601,Y 134.3658,Z 167,A 83.608,B 10.9309,C 0.0153,E1 10.9498,E2 367.2757} C_DIS
LIN {X 17.4603,Y 133.9982,Z 167,A 82.3316,B 10.9309,C 0.0146,E1 10.9534,E2 368.546} C_DIS
LIN {X 20.2244,Y 133.6097,Z 167,A 81.2643,B 10.9309,C 0.0124,E1 10.9563,E2 369.599} C_DIS
LIN {X 23.7897,Y 133.0203,Z 167,A 79.5532,B 10.9309,C 0.0172,E1 10.961,E2 371.331} C_DIS
LIN {X 27.8933,Y 132.2222,Z 167,A 77.7314,B 10.9309,C 0.0193,E1 10.966,E2 373.1583} C_DIS
LIN {X 31.3206,Y 131.4514,Z 167,A 76.4384,B 10.9309,C 0.0156,E1 10.9695,E2 374.4274} C_DIS
LIN {X 33.8954,Y 130.8124,Z 167,A 75.1846,B 10.9309,C 0.0194,E1 10.9729,E2 375.6965} C_DIS
LIN {X 37.689,Y 129.7688,Z 167,A 73.438,B 10.9309,C 0.0225,E1 10.9776,E2 377.4522} C_DIS
LIN {X 42.134,Y 128.3954,Z 167,A 71.5816,B 10.9309,C 0.0214,E1 10.9825,E2 379.2944} C_DIS
LIN {X 45.6189,Y 127.1977,Z 167,A 70.0137,B 10.9309,C 0.023,E1 10.9867,E2 380.8629} C_DIS
LIN {X 48.4961,Y 126.1296,Z 167,A 68.8657,B 10.9309,C 0.0206,E1 10.9896,E2 381.9923} C_DIS
LIN {X 50.8483,Y 125.1993,Z 167,A 67.5429,B 10.9309,C 0.0277,E1 10.9931,E2 383.3452} C_DIS
LIN {X 54.8574,Y 123.4952,Z 167,A 65.7962,B 10.9309,C 0.0274,E1 10.9976,E2 385.0797} C_DIS
LIN {X 57.9013,Y 122.0977,Z 167,A 64.5904,B 10.9309,C 0.0239,E1 11.0006,E2 386.2598} C_DIS
LIN {X 61.1067,Y 120.525,Z 167,A 62.6802,B 10.9309,C 0.0354,E1 11.0055,E2 388.2176} C_DIS
LIN {X 65.8657,Y 117.9944,Z 167,A 60.8117,B 10.9309,C 0.0284,E1 11.0099,E2 390.0363} C_DIS
LIN {X 70.0893,Y 115.535,Z 167,A 58.5121,B 10.9309,C 0.037,E1 11.0155,E2 392.3636} C_DIS
LIN {X 73.7861,Y 113.2099,Z 167,A 56.6684,B 10.9309,C 0.0396,E1 11.0199,E2 394.2066} C_DIS
LIN {X 77.1584,Y 110.9387,Z 167,A 54.7625,B 10.9309,C 0.0469,E1 11.0243,E2 396.1347} C_DIS
LIN {X 81.545,Y 107.7555,Z 167,A 52.8094,B 10.9309,C 0.0423,E1 11.0286,E2 398.0469} C_DIS
LIN {X 84.8401,Y 105.1806,Z 167,A 50.9798,B 10.9309,C 0.0468,E1 11.0326,E2 399.8837} C_DIS
LIN {X 87.9707,Y 102.577,Z 167,A 49.1566,B 10.9308,C 0.0524,E1 11.0365,E2 401.7191} C_DIS
LIN {X 91.2338,Y 99.6859,Z 167,A 47.326,B 10.9308,C 0.0555,E1 11.0403,E2 403.5483} C_DIS
LIN {X 94.571,Y 96.5253,Z 167,A 45.4304,B 10.9308,C 0.0581,E1 11.0441,E2 405.4381} C_DIS
LIN {X 97.7499,Y 93.3046,Z 167,A 43.5513,B 10.9308,C 0.061,E1 11.0478,E2 407.3132} C_DIS
LIN {X 100.6255,Y 90.196,Z 167,A 41.7439,B 10.9308,C 0.0651,E1 11.0512,E2 409.1228} C_DIS
LIN {X 103.588,Y 86.7776,Z 167,A 39.8258,B 10.9307,C 0.0694,E1 11.0547,E2 411.0419} C_DIS
LIN {X 106.8189,Y 82.7679,Z 167,A 37.6811,B 10.9307,C 0.0733,E1 11.0584,E2 413.183} C_DIS
LIN {X 109.5394,Y 79.1326,Z 167,A 35.8743,B 10.9307,C 0.0748,E1 11.0614,E2 414.9766} C_DIS
LIN {X 111.8952,Y 75.7646,Z 167,A 34.0693,B 10.9307,C 0.0805,E1 11.0642,E2 416.7901} C_DIS
LIN {X 114.2096,Y 72.2288,Z 167,A 32.3179,B 10.9306,C 0.0838,E1 11.0669,E2 418.5378} C_DIS
LIN {X 116.2932,Y 68.8249,Z 167,A 30.4844,B 10.9306,C 0.0917,E1 11.0695,E2 420.3895} C_DIS
LIN {X 118.7399,Y 64.5111,Z 167,A 28.5373,B 10.9306,C 0.093,E1 11.0722,E2 422.319} C_DIS
LIN {X 120.7943,Y 60.5777,Z 167,A 26.7794,B 10.9306,C 0.0947,E1 11.0744,E2 424.0633} C_DIS
LIN {X 122.3583,Y 57.3517,Z 167,A 25.2007,B 10.9305,C 0.1002,E1 11.0763,E2 425.6502} C_DIS
LIN {X 123.8433,Y 54.0681,Z 167,A 23.7647,B 10.9305,C 0.1018,E1 11.0779,E2 427.0761} C_DIS
LIN {X 125.0311,Y 51.2656,Z 167,A 22.5053,B 10.9305,C 0.1045,E1 11.0793,E2 428.3327} C_DIS
LIN {X 125.901,Y 49.0841,Z 167,A 21.0713,B 10.9303,C 0.1185,E1 11.0808,E2 429.8207} C_DIS
LIN {X 127.3409,Y 45.2217,Z 167,A 19.7205,B 10.9303,C 0.113,E1 11.082,E2 431.1247} C_DIS
LIN {X 129.5229,Y 38.529,Z 167,A 16.778,B 10.9303,C 0.1202,E1 11.0845,E2 434.0646} C_DIS
LIN {X 130.5075,Y 35.0453,Z 167,A 15.3064,B 10.9303,C 0.1229,E1 11.0856,E2 435.5297} C_DIS
LIN {X 131.3498,Y 31.7422,Z 167,A 14.0478,B 10.9303,C 0.1221,E1 11.0864,E2 436.7667} C_DIS
LIN {X 131.911,Y 29.3329,Z 167,A 12.7065,B 10.9301,C 0.1328,E1 11.0873,E2 438.1449} C_DIS
LIN {X 132.7371,Y 25.3222,Z 167,A 11.139,B 10.9301,C 0.1333,E1 11.0881,E2 439.6932} C_DIS
LIN {X 133.3828,Y 21.6729,Z 167,A 9.4471,B 10.9301,C 0.141,E1 11.0889,E2 441.4014} C_DIS
LIN {X 133.9217,Y 18.0444,Z 167,A 8.1923,B 10.9301,C 0.1376,E1 11.0894,E2 442.6209} C_DIS
LIN {X 134.3581,Y 14.432,Z 167,A 6.5318,B 10.93,C 0.1452,E1 11.0899,E2 444.2973} C_DIS
LIN {X 134.7237,Y 10.5056,Z 167,A 4.7482,B 10.9299,C 0.153,E1 11.0903,E2 446.0962} C_DIS
LIN {X 134.9948,Y 6.1057,Z 167,A 2.9376,B 10.9299,C 0.157,E1 11.0906,E2 447.9016} C_DIS
LIN {X 135.1173,Y 1.954,Z 167,A 1.1825,B 10.9297,C 0.162,E1 11.0907,E2 449.6577} C_DIS
LIN {X 135.1148,Y -2.1054,Z 167,A -0.4096,B 10.9297,C 0.1636,E1 11.0907,E2 451.2357} C_DIS
LIN {X 134.9576,Y -6.8452,Z 167,A -2.589,B 10.9295,C 0.174,E1 11.0904,E2 453.4379} C_DIS
LIN {X 134.6276,Y -11.6568,Z 167,A -4.5002,B 10.9295,C 0.1764,E1 11.09,E2 455.3348} C_DIS
LIN {X 134.1996,Y -15.8388,Z 167,A -6.1455,B 10.9295,C 0.1781,E1 11.0895,E2 456.9652} C_DIS
LIN {X 133.7723,Y -19.1142,Z 167,A -7.5426,B 10.9295,C 0.1821,E1 11.089,E2 458.3634} C_DIS
LIN {X 133.2623,Y -22.3954,Z 167,A -8.9925,B 10.9293,C 0.1873,E1 11.0883,E2 459.82} C_DIS
LIN {X 132.4424,Y -26.8213,Z 167,A -10.6234,B 10.9293,C 0.1855,E1 11.0875,E2 461.4188} C_DIS
LIN {X 131.9144,Y -29.3182,Z 167,A -12.0358,B 10.9292,C 0.1974,E1 11.0866,E2 462.8732} C_DIS
LIN {X 131.0759,Y -32.8571,Z 167,A -13.5892,B 10.9291,C 0.2021,E1 11.0856,E2 464.4297} C_DIS
LIN {X 129.6593,Y -38.063,Z 167,A -15.6083,B 10.9291,C 0.2015,E1 11.0841,E2 466.4182} C_DIS
LIN {X 128.7822,Y -40.9326,Z 167,A -16.7218,B 10.9291,C 0.201,E1 11.0832,E2 467.5134} C_DIS
LIN {X 128.0743,Y -43.0982,Z 167,A -18.0905,B 10.9288,C 0.2143,E1 11.0819,E2 468.933} C_DIS
LIN {X 125.1204,Y -51.044,Z 167,A -21.5431,B 10.9288,C 0.2206,E1 11.0785,E2 472.3722} C_DIS
LIN {X 123.5679,Y -54.6947,Z 167,A -23.2006,B 10.9286,C 0.2245,E1 11.0767,E2 474.0286} C_DIS
LIN {X 122.1875,Y -57.7135,Z 167,A -24.3651,B 10.9286,C 0.222,E1 11.0753,E2 475.1647} C_DIS
LIN {X 121.0175,Y -60.1264,Z 167,A -25.5332,B 10.9286,C 0.2258,E1 11.0739,E2 476.3379} C_DIS
LIN {X 119.3307,Y -63.4105,Z 167,A -27.2062,B 10.9285,C 0.2328,E1 11.0717,E2 478.0261} C_DIS
LIN {X 117.3038,Y -67.0869,Z 167,A -28.9937,B 10.9284,C 0.2377,E1 11.0692,E2 479.8165} C_DIS
LIN {X 114.9755,Y -71.0043,Z 167,A -30.9293,B 10.9283,C 0.2427,E1 11.0664,E2 481.7547} C_DIS
LIN {X 112.5772,Y -74.7482,Z 167,A -32.7713,B 10.9282,C 0.2464,E1 11.0636,E2 483.5935} C_DIS
LIN {X 110.0987,Y -78.3528,Z 167,A -34.5847,B 10.9281,C 0.2499,E1 11.0607,E2 485.4038} C_DIS
LIN {X 107.5191,Y -81.8568,Z 167,A -36.4077,B 10.9281,C 0.2538,E1 11.0577,E2 487.2262} C_DIS
LIN {X 104.9251,Y -85.1569,Z 167,A -39.0996,B 10.9273,C 0.2814,E1 11.0528,E2 490.0321} C_DIS
LIN {X 100.266,Y -90.5959,Z 167,A -41.2024,B 10.9278,C 0.2644,E1 11.0491,E2 492.0236} C_DIS
LIN {X 97.1549,Y -93.9241,Z 167,A -43.0405,B 10.9278,C 0.2663,E1 11.0455,E2 493.8522} C_DIS
LIN {X 94.1276,Y -96.9578,Z 167,A -44.972,B 10.9275,C 0.2731,E1 11.0417,E2 495.7998} C_DIS
LIN {X 89.0841,Y -101.6116,Z 167,A -47.7832,B 10.9275,C 0.2766,E1 11.0359,E2 498.6018} C_DIS
LIN {X 85.78,Y -104.416,Z 167,A -49.5901,B 10.9274,C 0.2795,E1 11.032,E2 500.4068} C_DIS
LIN {X 82.2995,Y -107.1805,Z 167,A -51.5652,B 10.9272,C 0.2853,E1 11.0276,E2 502.395} C_DIS
LIN {X 78.0755,Y -110.2954,Z 167,A -53.4558,B 10.9273,C 0.2809,E1 11.0234,E2 504.2463} C_DIS
LIN {X 70.2802,Y -115.4195,Z 167,A -57.6164,B 10.927,C 0.2929,E1 11.0137,E2 508.4364} C_DIS
LIN {X 66.3713,Y -117.7102,Z 167,A -59.491,B 10.927,C 0.2947,E1 11.0091,E2 510.307} C_DIS
LIN {X 63.03,Y -119.5305,Z 167,A -61.0518,B 10.927,C 0.2958,E1 11.0053,E2 511.8627} C_DIS
LIN {X 59.7827,Y -121.187,Z 167,A -62.4624,B 10.927,C 0.2947,E1 11.0018,E2 513.2578} C_DIS
LIN {X 56.924,Y -122.556,Z 167,A -63.6729,B 10.927,C 0.2932,E1 10.9988,E2 514.4529} C_DIS
LIN {X 54.6486,Y -123.5886,Z 167,A -65.0757,B 10.9268,C 0.3031,E1 10.9951,E2 515.8993} C_DIS
LIN {X 50.85,Y -125.1986,Z 167,A -66.5122,B 10.9269,C 0.2976,E1 10.9915,E2 517.2984} C_DIS
LIN {X 46.2743,Y -126.9614,Z 167,A -68.6319,B 10.9269,C 0.301,E1 10.9859,E2 519.425} C_DIS
LIN {X 38.8465,Y -129.4287,Z 167,A -72.1574,B 10.9266,C 0.3095,E1 10.9765,E2 522.9789} C_DIS
LIN {X 35.7035,Y -130.3307,Z 167,A -73.5349,B 10.9266,C 0.3106,E1 10.9728,E2 524.3563} C_DIS
LIN {X 32.2257,Y -131.2333,Z 167,A -74.8314,B 10.9266,C 0.3063,E1 10.9694,E2 525.6258} C_DIS
LIN {X 29.851,Y -131.7927,Z 167,A -75.8852,B 10.9266,C 0.3076,E1 10.9665,E2 526.6826} C_DIS
LIN {X 26.5068,Y -132.5064,Z 167,A -77.5374,B 10.9265,C 0.3136,E1 10.9619,E2 528.361} C_DIS
LIN {X 22.4827,Y -133.2477,Z 167,A -79.1204,B 10.9265,C 0.311,E1 10.9576,E2 529.9262} C_DIS
LIN {X 19.3365,Y -133.7405,Z 167,A -80.3845,B 10.9265,C 0.3097,E1 10.9541,E2 531.1805} C_DIS
LIN {X 16.7925,Y -134.0857,Z 167,A -81.7194,B 10.9264,C 0.3162,E1 10.9503,E2 532.5466} C_DIS
LIN {X 13.0688,Y -134.4977,Z 167,A -83.1641,B 10.9264,C 0.3134,E1 10.9464,E2 533.9744} C_DIS
LIN {X 9.4278,Y -134.8024,Z 167,A -84.8355,B 10.9264,C 0.3169,E1 10.9417,E2 535.6618} C_DIS
LIN {X 5.8104,Y -135.0072,Z 167,A -86.1235,B 10.9265,C 0.3114,E1 10.9382,E2 536.9198} C_DIS
LIN {X 2.1894,Y -135.1134,Z 167,A -87.8243,B 10.9265,C 0.3156,E1 10.9334,E2 538.6419} C_DIS
LIN {X 2.1894,Y -135.1134,Z 167,A -87.8243,B 10.9265,C 0.3156,E1 10.9334,E2 538.6419} C_DIS
Enddeposition()
LIN {X 0.9784,Y -136.0431,Z 167,A -87.9766,B 10.839,C 0.3174,E1 10.8456,E2 538.8102} C_DIS
Startdeposition()
$VEL.CP = VEL_PRINT
LIN {X 4.5393,Y -135.9731,Z 167,A -86.1079,B 10.8393,C 0.3084,E1 10.8509,E2 536.8944} C_DIS
LIN {X 8.1419,Y -135.803,Z 167,A -84.5559,B 10.8393,C 0.3071,E1 10.8553,E2 535.3373} C_DIS
LIN {X 12.2246,Y -135.4985,Z 167,A -82.8633,B 10.8393,C 0.3073,E1 10.86,E2 533.6478} C_DIS
LIN {X 15.3344,Y -135.1819,Z 167,A -81.5645,B 10.8393,C 0.3071,E1 10.8636,E2 532.3504} C_DIS
LIN {X 18.5079,Y -134.7838,Z 167,A -80.1385,B 10.8393,C 0.3045,E1 10.8675,E2 530.9136} C_DIS
LIN {X 22.0906,Y -134.2413,Z 167,A -78.66,B 10.8393,C 0.3047,E1 10.8716,E2 529.44} C_DIS
LIN {X 25.2396,Y -133.685,Z 167,A -77.5085,B 10.8393,C 0.3086,E1 10.8747,E2 528.3124} C_DIS
LIN {X 27.9185,Y -133.1534,Z 167,A -76.1837,B 10.8394,C 0.3036,E1 10.8784,E2 526.9649} C_DIS
LIN {X 31.0879,Y -132.4493,Z 167,A -74.6851,B 10.8395,C 0.2992,E1 10.8825,E2 525.4486} C_DIS
LIN {X 34.3082,Y -131.6516,Z 167,A -73.443,B 10.8395,C 0.3019,E1 10.8858,E2 524.2252} C_DIS
LIN {X 37.538,Y -130.767,Z 167,A -72.0769,B 10.8395,C 0.3017,E1 10.8895,E2 522.8636} C_DIS
LIN {X 40.6068,Y -129.8475,Z 167,A -70.674,B 10.8395,C 0.299,E1 10.8933,E2 521.4529} C_DIS
LIN {X 43.8205,Y -128.7981,Z 167,A -69.1636,B 10.8396,C 0.2954,E1 10.8973,E2 519.9305} C_DIS
LIN {X 47.4608,Y -127.4995,Z 167,A -67.8627,B 10.8395,C 0.3017,E1 10.9006,E2 518.6695} C_DIS
LIN {X 50.0788,Y -126.4966,Z 167,A -66.4766,B 10.8396,C 0.2952,E1 10.9043,E2 517.2566} C_DIS
LIN {X 53.211,Y -125.2113,Z 167,A -65.0576,B 10.8396,C 0.2936,E1 10.9079,E2 515.8372} C_DIS
LIN {X 56.3713,Y -123.8203,Z 167,A -63.6108,B 10.8397,C 0.2918,E1 10.9116,E2 514.3901} C_DIS
LIN {X 59.4639,Y -122.3652,Z 167,A -62.1793,B 10.8397,C 0.29,E1 10.9152,E2 512.9584} C_DIS
LIN {X 62.4865,Y -120.85,Z 167,A -60.7568,B 10.8398,C 0.288,E1 10.9188,E2 511.5348} C_DIS
LIN {X 66.0678,Y -118.9293,Z 167,A -59.0028,B 10.8399,C 0.2843,E1 10.9231,E2 509.7738} C_DIS
LIN {X 69.3294,Y -117.0584,Z 167,A -57.4978,B 10.8399,C 0.2838,E1 10.9267,E2 508.2773} C_DIS
LIN {X 72.2484,Y -115.2799,Z 167,A -56.0608,B 10.8399,C 0.2815,E1 10.9301,E2 506.8393} C_DIS
LIN {X 75.1751,Y -113.393,Z 167,A -54.5979,B 10.8401,C 0.2791,E1 10.9335,E2 505.3754} C_DIS
LIN {X 78.5873,Y -111.0548,Z 167,A -52.8481,B 10.8401,C 0.2758,E1 10.9376,E2 503.6229} C_DIS
LIN {X 81.623,Y -108.8437,Z 167,A -51.3082,B 10.8401,C 0.2739,E1 10.941,E2 502.0867} C_DIS
LIN {X 84.4016,Y -106.7035,Z 167,A -49.8507,B 10.8402,C 0.2716,E1 10.9442,E2 500.6302} C_DIS
LIN {X 87.5552,Y -104.1306,Z 167,A -48.0832,B 10.8404,C 0.2669,E1 10.948,E2 498.8542} C_DIS
LIN {X 90.7872,Y -101.3251,Z 167,A -46.299,B 10.8404,C 0.2637,E1 10.9518,E2 497.0704} C_DIS
LIN {X 93.6787,Y -98.6589,Z 167,A -44.7185,B 10.8404,C 0.2622,E1 10.955,E2 495.4979} C_DIS
LIN {X 96.2195,Y -96.1825,Z 167,A -43.2393,B 10.8405,C 0.2594,E1 10.9579,E2 494.0189} C_DIS
LIN {X 98.8493,Y -93.4769,Z 167,A -41.7313,B 10.8405,C 0.258,E1 10.9608,E2 492.5195} C_DIS
LIN {X 101.0498,Y -91.0945,Z 167,A -40.3154,B 10.8407,C 0.2536,E1 10.9635,E2 491.0957} C_DIS
LIN {X 103.3885,Y -88.4312,Z 167,A -38.839,B 10.8407,C 0.2506,E1 10.9662,E2 489.6198} C_DIS
LIN {X 105.6219,Y -85.7513,Z 167,A -37.3862,B 10.8408,C 0.2476,E1 10.9688,E2 488.1675} C_DIS
LIN {X 107.8641,Y -82.9129,Z 167,A -35.9018,B 10.8408,C 0.245,E1 10.9713,E2 486.6863} C_DIS
LIN {X 109.916,Y -80.1731,Z 167,A -34.4557,B 10.841,C 0.2414,E1 10.9737,E2 485.2381} C_DIS
LIN {X 111.9257,Y -77.3428,Z 167,A -33.0043,B 10.841,C 0.238,E1 10.976,E2 483.7863} C_DIS
LIN {X 114.1985,Y -73.9448,Z 167,A -31.2687,B 10.8411,C 0.2333,E1 10.9787,E2 482.0471} C_DIS
LIN {X 116.3058,Y -70.584,Z 167,A -29.5555,B 10.8412,C 0.2279,E1 10.9812,E2 480.3266} C_DIS
LIN {X 118.6631,Y -66.5445,Z 167,A -27.6635,B 10.8413,C 0.2248,E1 10.9838,E2 478.4421} C_DIS
LIN {X 120.85,Y -62.4865,Z 167,A -25.8007,B 10.8413,C 0.2218,E1 10.9863,E2 476.5872} C_DIS
LIN {X 122.3877,Y -59.4182,Z 167,A -24.3746,B 10.8414,C 0.2184,E1 10.988,E2 475.1619} C_DIS
LIN {X 123.8623,Y -56.279,Z 167,A -22.9339,B 10.8415,C 0.215,E1 10.9897,E2 473.722} C_DIS
LIN {X 125.3123,Y -52.9692,Z 167,A -21.5087,B 10.8415,C 0.2134,E1 10.9913,E2 472.3072} C_DIS
LIN {X 126.5148,Y -50.0321,Z 167,A -20.1337,B 10.8416,C 0.2087,E1 10.9927,E2 470.9259} C_DIS
LIN {X 127.6976,Y -46.9319,Z 167,A -18.7376,B 10.8416,C 0.2048,E1 10.9941,E2 469.5284} C_DIS
LIN {X 128.8144,Y -43.7735,Z 167,A -17.3293,B 10.8418,C 0.2009,E1 10.9954,E2 468.1188} C_DIS
LIN {X 129.8785,Y -40.5054,Z 167,A -15.8414,B 10.8418,C 0.1957,E1 10.9966,E2 466.6241} C_DIS
LIN {X 130.8001,Y -37.4245,Z 167,A -14.5897,B 10.8418,C 0.1946,E1 10.9976,E2 465.3839} C_DIS
LIN {X 131.6642,Y -34.261,Z 167,A -13.2078,B 10.842,C 0.1907,E1 10.9986,E2 464.0003} C_DIS
LIN {X 132.4493,Y -31.0879,Z 167,A -11.8516,B 10.842,C 0.1872,E1 10.9995,E2 462.6453} C_DIS
LIN {X 133.2268,Y -27.558,Z 167,A -10.5051,B 10.842,C 0.1875,E1 11.0003,E2 461.3191} C_DIS
LIN {X 133.7859,Y -24.7089,Z 167,A -9.1657,B 10.8421,C 0.1809,E1 11.001,E2 459.9637} C_DIS
LIN {X 134.3228,Y -21.6025,Z 167,A -7.8575,B 10.8421,C 0.1775,E1 11.0016,E2 458.6565} C_DIS
LIN {X 134.8282,Y -18.1733,Z 167,A -6.3533,B 10.8423,C 0.172,E1 11.0021,E2 457.1452} C_DIS
LIN {X 135.2271,Y -14.9138,Z 167,A -5.1063,B 10.8423,C 0.1716,E1 11.0025,E2 455.9137} C_DIS
LIN {X 135.4985,Y -12.2246,Z 167,A -3.921,B 10.8423,C 0.167,E1 11.0029,E2 454.7214} C_DIS
LIN {X 135.7447,Y -9.0884,Z 167,A -2.6508,B 10.8423,C 0.1646,E1 11.0031,E2 453.4565} C_DIS
LIN {X 135.9153,Y -6.0197,Z 167,A -1.3597,B 10.8424,C 0.1609,E1 11.0033,E2 452.1646} C_DIS
LIN {X 136.0233,Y -2.5376,Z 167,A 0.0122,B 10.8424,C 0.1591,E1 11.0033,E2 450.803} C_DIS
LIN {X 136.0489,Y 0,Z 167,A 1.156,B 10.8425,C 0.154,E1 11.0034,E2 449.6488} C_DIS
LIN {X 136.0153,Y 3.0197,Z 167,A 2.5202,B 10.8426,C 0.1478,E1 11.0034,E2 448.2717} C_DIS
LIN {X 135.9113,Y 6.1106,Z 167,A 3.6652,B 10.8426,C 0.1482,E1 11.0032,E2 447.1451} C_DIS
LIN {X 135.7418,Y 9.1341,Z 167,A 5.0705,B 10.8427,C 0.141,E1 11.003,E2 445.7223} C_DIS
LIN {X 135.3444,Y 13.8235,Z 167,A 6.8842,B 10.8427,C 0.1397,E1 11.0025,E2 443.9278} C_DIS
LIN {X 134.9956,Y 16.8958,Z 167,A 8.2055,B 10.8427,C 0.1354,E1 11.0021,E2 442.6028} C_DIS
LIN {X 134.559,Y 20.077,Z 167,A 9.507,B 10.8428,C 0.1328,E1 11.0015,E2 441.3063} C_DIS
LIN {X 133.9617,Y 23.7265,Z 167,A 11.0482,B 10.8428,C 0.1287,E1 11.0008,E2 439.7656} C_DIS
LIN {X 133.4238,Y 26.5896,Z 167,A 12.1808,B 10.8428,C 0.1277,E1 11.0002,E2 438.6437} C_DIS
LIN {X 132.8007,Y 29.5497,Z 167,A 13.6284,B 10.843,C 0.1195,E1 10.9994,E2 437.1733} C_DIS
LIN {X 131.955,Y 33.1154,Z 167,A 15.0985,B 10.843,C 0.1171,E1 10.9984,E2 435.7109} C_DIS
LIN {X 131.1283,Y 36.2512,Z 167,A 16.4494,B 10.843,C 0.1136,E1 10.9974,E2 434.3607} C_DIS
LIN {X 130.3327,Y 39.0213,Z 167,A 17.6103,B 10.843,C 0.1116,E1 10.9965,E2 433.2055} C_DIS
LIN {X 129.3257,Y 42.2381,Z 167,A 19.1364,B 10.8431,C 0.1049,E1 10.9952,E2 431.6648} C_DIS
LIN {X 128.2496,Y 45.4009,Z 167,A 20.404,B 10.8431,C 0.1047,E1 10.994,E2 430.4136} C_DIS
LIN {X 127.1076,Y 48.507,Z 167,A 21.7816,B 10.8431,C 0.1013,E1 10.9927,E2 429.0369} C_DIS
LIN {X 125.8645,Y 51.647,Z 167,A 23.1877,B 10.8431,C 0.0979,E1 10.9912,E2 427.6317} C_DIS
LIN {X 124.3427,Y 55.2049,Z 167,A 24.7013,B 10.8431,C 0.0966,E1 10.9895,E2 426.1312} C_DIS
LIN {X 123.1033,Y 57.9205,Z 167,A 26.0416,B 10.8432,C 0.0911,E1 10.9879,E2 424.7797} C_DIS
LIN {X 121.6061,Y 61.0011,Z 167,A 27.5901,B 10.8432,C 0.0846,E1 10.986,E2 423.217} C_DIS
LIN {X 119.6419,Y 64.7696,Z 167,A 29.245,B 10.8432,C 0.0835,E1 10.9839,E2 421.5777} C_DIS
LIN {X 117.659,Y 68.3043,Z 167,A 30.9677,B 10.8433,C 0.0788,E1 10.9815,E2 419.8518} C_DIS
LIN {X 115.739,Y 71.5105,Z 167,A 32.6062,B 10.8433,C 0.0733,E1 10.9791,E2 418.2043} C_DIS
LIN {X 113.3791,Y 75.196,Z 167,A 34.3065,B 10.8433,C 0.0725,E1 10.9765,E2 416.5206} C_DIS
LIN {X 111.2337,Y 78.3337,Z 167,A 35.9753,B 10.8434,C 0.0669,E1 10.9738,E2 414.8425} C_DIS
LIN {X 108.8041,Y 81.6754,Z 167,A 37.5941,B 10.8434,C 0.066,E1 10.9712,E2 413.2378} C_DIS
LIN {X 106.7035,Y 84.4016,Z 167,A 39.0392,B 10.8434,C 0.0628,E1 10.9687,E2 411.7924} C_DIS
LIN {X 104.5058,Y 87.1081,Z 167,A 40.6153,B 10.8434,C 0.0568,E1 10.9659,E2 410.2023} C_DIS
LIN {X 101.6194,Y 90.4586,Z 167,A 42.3367,B 10.8434,C 0.0564,E1 10.9627,E2 408.4975} C_DIS
LIN {X 99.263,Y 93.0384,Z 167,A 43.9224,B 10.8434,C 0.0503,E1 10.9597,E2 406.8971} C_DIS
LIN {X 96.124,Y 96.2776,Z 167,A 45.7936,B 10.8435,C 0.0472,E1 10.956,E2 405.0286} C_DIS
LIN {X 93.0192,Y 99.2808,Z 167,A 47.4847,B 10.8435,C 0.0468,E1 10.9526,E2 403.3526} C_DIS
LIN {X 90.0921,Y 101.9436,Z 167,A 49.2036,B 10.8435,C 0.0423,E1 10.949,E2 401.6266} C_DIS
LIN {X 87.088,Y 104.5225,Z 167,A 50.8044,B 10.8435,C 0.0409,E1 10.9456,E2 400.0336} C_DIS
LIN {X 84.3812,Y 106.7197,Z 167,A 52.28,B 10.8435,C 0.0381,E1 10.9424,E2 398.5567} C_DIS
LIN {X 81.2921,Y 109.0903,Z 167,A 53.9571,B 10.8435,C 0.0343,E1 10.9387,E2 396.8746} C_DIS
LIN {X 78.0386,Y 111.4416,Z 167,A 55.5395,B 10.8435,C 0.0343,E1 10.9351,E2 395.3052} C_DIS
LIN {X 75.1751,Y 113.393,Z 167,A 57.087,B 10.8435,C 0.0297,E1 10.9315,E2 393.7466} C_DIS
LIN {X 71.4659,Y 115.7664,Z 167,A 58.8201,B 10.8435,C 0.0299,E1 10.9274,E2 392.0281} C_DIS
LIN {X 68.536,Y 117.5249,Z 167,A 60.3702,B 10.8435,C 0.0251,E1 10.9237,E2 390.4642} C_DIS
LIN {X 64.7696,Y 119.6419,Z 167,A 62.2014,B 10.8435,C 0.0223,E1 10.9192,E2 388.6315} C_DIS
LIN {X 60.9556,Y 121.6293,Z 167,A 63.8678,B 10.8435,C 0.0235,E1 10.9151,E2 386.9827} C_DIS
LIN {X 57.6667,Y 123.2213,Z 167,A 65.4658,B 10.8435,C 0.0202,E1 10.911,E2 385.3774} C_DIS
LIN {X 54.7006,Y 124.5673,Z 167,A 66.7501,B 10.8435,C 0.0208,E1 10.9078,E2 384.1038} C_DIS
LIN {X 51.6004,Y 125.8833,Z 167,A 68.169,B 10.8435,C 0.0192,E1 10.9041,E2 382.6849} C_DIS
LIN {X 48.507,Y 127.1076,Z 167,A 69.5621,B 10.8435,C 0.018,E1 10.9005,E2 381.2929} C_DIS
LIN {X 45.354,Y 128.2665,Z 167,A 70.9686,B 10.8435,C 0.0169,E1 10.8968,E2 379.8875} C_DIS
LIN {X 42.1439,Y 129.3565,Z 167,A 72.4813,B 10.8436,C 0.0136,E1 10.8928,E2 378.3646} C_DIS
LIN {X 39.0213,Y 130.3327,Z 167,A 73.7595,B 10.8436,C 0.0148,E1 10.8894,E2 377.0988} C_DIS
LIN {X 35.7187,Y 131.2755,Z 167,A 75.1489,B 10.8436,C 0.0151,E1 10.8857,E2 375.7167} C_DIS
LIN {X 32.6269,Y 132.0783,Z 167,A 76.6611,B 10.8436,C 0.0102,E1 10.8815,E2 374.1843} C_DIS
LIN {X 28.9302,Y 132.935,Z 167,A 78.121,B 10.8436,C 0.0126,E1 10.8776,E2 372.7416} C_DIS
LIN {X 25.8313,Y 133.5719,Z 167,A 79.4382,B 10.8436,C 0.0122,E1 10.874,E2 371.4265} C_DIS
LIN {X 23.131,Y 134.0678,Z 167,A 80.5901,B 10.8436,C 0.0118,E1 10.8708,E2 370.2756} C_DIS
LIN {X 20.0302,Y 134.5662,Z 167,A 81.9427,B 10.8436,C 0.0106,E1 10.8671,E2 368.9197} C_DIS
LIN {X 16.4424,Y 135.0497,Z 167,A 83.4824,B 10.8436,C 0.0097,E1 10.8628,E2 367.3786} C_DIS
LIN {X 13.0471,Y 135.4195,Z 167,A 84.7346,B 10.8436,C 0.0137,E1 10.8594,E2 366.1496} C_DIS
LIN {X 10.6309,Y 135.6326,Z 167,A 85.8982,B 10.8436,C 0.0102,E1 10.8561,E2 364.9692} C_DIS
LIN {X 7.5968,Y 135.8366,Z 167,A 87.1924,B 10.8436,C 0.0097,E1 10.8525,E2 363.6738} C_DIS
LIN {X 4.4941,Y 135.9743,Z 167,A 88.61,B 10.8436,C 0.0071,E1 10.8485,E2 362.2434} C_DIS
LIN {X 0.7132,Y 136.0449,Z 167,A 89.9713,B 10.8436,C 0.0124,E1 10.8448,E2 360.911} C_DIS
LIN {X -3.0197,Y 136.0153,Z 167,A 91.6462,B 10.8436,C 0.0102,E1 10.8401,E2 359.2244} C_DIS
LIN {X -6.1106,Y 135.9113,Z 167,A 92.9346,B 10.8436,C 0.0107,E1 10.8365,E2 357.9383} C_DIS
LIN {X -9.1341,Y 135.7418,Z 167,A 94.3868,B 10.8436,C 0.007,E1 10.8324,E2 356.4653} C_DIS
LIN {X -12.9871,Y 135.4253,Z 167,A 95.8334,B 10.8436,C 0.0116,E1 10.8284,E2 355.0416} C_DIS
LIN {X -16.8958,Y 134.9956,Z 167,A 97.5444,B 10.8436,C 0.011,E1 10.8237,E2 353.3249} C_DIS
LIN {X -20.077,Y 134.559,Z 167,A 98.8665,B 10.8436,C 0.0123,E1 10.82,E2 352.0073} C_DIS
LIN {X -23.6108,Y 133.9824,Z 167,A 100.3795,B 10.8436,C 0.013,E1 10.8159,E2 350.4946} C_DIS
LIN {X -26.3833,Y 133.4658,Z 167,A 101.574,B 10.8436,C 0.0136,E1 10.8126,E2 349.3001} C_DIS
LIN {X -29.5497,Y 132.8007,Z 167,A 102.9428,B 10.8436,C 0.0143,E1 10.8088,E2 347.9314} C_DIS
LIN {X -33.0443,Y 131.973,Z 167,A 104.5357,B 10.8436,C 0.0137,E1 10.8045,E2 346.3297} C_DIS
LIN {X -35.8952,Y 131.2278,Z 167,A 105.7287,B 10.8436,C 0.0157,E1 10.8013,E2 345.1435} C_DIS
LIN {X -39.0213,Y 130.3327,Z 167,A 107.2242,B 10.8436,C 0.0141,E1 10.7972,E2 343.6336} C_DIS
LIN {X -42.2381,Y 129.3257,Z 167,A 108.5338,B 10.8436,C 0.0179,E1 10.7938,E2 342.3385} C_DIS
LIN {X -45.4009,Y 128.2496,Z 167,A 109.9492,B 10.8436,C 0.0191,E1 10.7901,E2 340.9232} C_DIS
LIN {X -48.7642,Y 127.0077,Z 167,A 111.3644,B 10.8436,C 0.0228,E1 10.7864,E2 339.5207} C_DIS
LIN {X -51.647,Y 125.8645,Z 167,A 112.7835,B 10.8436,C 0.0219,E1 10.7827,E2 338.089} C_DIS
LIN {X -54.7706,Y 124.537,Z 167,A 114.241,B 10.8436,C 0.023,E1 10.779,E2 336.6292} C_DIS
LIN {X -58.1673,Y 122.9854,Z 167,A 115.8131,B 10.8436,C 0.025,E1 10.775,E2 335.0585} C_DIS
LIN {X -61.0011,Y 121.6061,Z 167,A 117.1241,B 10.8436,C 0.0271,E1 10.7717,E2 333.7506} C_DIS
LIN {X -64.033,Y 120.0377,Z 167,A 118.5921,B 10.8436,C 0.0285,E1 10.7681,E2 332.2802} C_DIS
LIN {X -67.0579,Y 118.3744,Z 167,A 120.0573,B 10.8436,C 0.0304,E1 10.7645,E2 330.8149} C_DIS
LIN {X -70.5533,Y 116.3244,Z 167,A 121.8108,B 10.8436,C 0.0321,E1 10.7603,E2 329.0572} C_DIS
LIN {X -73.7168,Y 114.3465,Z 167,A 123.362,B 10.8436,C 0.035,E1 10.7566,E2 327.5099} C_DIS
LIN {X -76.6444,Y 112.4051,Z 167,A 124.9827,B 10.8436,C 0.0345,E1 10.7528,E2 325.8735} C_DIS
LIN {X -80.3083,Y 109.8169,Z 167,A 126.8082,B 10.8436,C 0.0392,E1 10.7487,E2 324.0576} C_DIS
LIN {X -83.7117,Y 107.2456,Z 167,A 128.5731,B 10.8436,C 0.0431,E1 10.7448,E2 322.2983} C_DIS
LIN {X -86.4314,Y 105.0661,Z 167,A 130.0546,B 10.8436,C 0.0456,E1 10.7416,E2 320.8166} C_DIS
LIN {X -89.5612,Y 102.4105,Z 167,A 131.878,B 10.8436,C 0.047,E1 10.7377,E2 318.9834} C_DIS
LIN {X -92.3942,Y 99.8628,Z 167,A 133.42,B 10.8435,C 0.0516,E1 10.7346,E2 317.4506} C_DIS
LIN {X -94.9478,Y 97.4382,Z 167,A 134.9252,B 10.8435,C 0.0542,E1 10.7315,E2 315.9443} C_DIS
LIN {X -97.4564,Y 94.929,Z 167,A 136.5454,B 10.8435,C 0.0547,E1 10.7283,E2 314.3103} C_DIS
LIN {X -100.5482,Y 91.6474,Z 167,A 138.3166,B 10.8435,C 0.0615,E1 10.725,E2 312.5566} C_DIS
LIN {X -102.8148,Y 89.0976,Z 167,A 139.7979,B 10.8435,C 0.0638,E1 10.7223,E2 311.0715} C_DIS
LIN {X -105.0827,Y 86.4112,Z 167,A 141.2872,B 10.8435,C 0.0671,E1 10.7196,E2 309.5828} C_DIS
LIN {X -107.473,Y 83.4185,Z 167,A 143.0178,B 10.8434,C 0.0684,E1 10.7166,E2 307.8395} C_DIS
LIN {X -110.2192,Y 79.7548,Z 167,A 144.9285,B 10.8434,C 0.0734,E1 10.7135,E2 305.9331} C_DIS
LIN {X -112.7672,Y 76.1096,Z 167,A 146.849,B 10.8434,C 0.077,E1 10.7104,E2 304.0088} C_DIS
LIN {X -114.8295,Y 72.9619,Z 167,A 148.3643,B 10.8433,C 0.0824,E1 10.7081,E2 302.5038} C_DIS
LIN {X -116.6421,Y 70.0278,Z 167,A 149.8409,B 10.8433,C 0.0856,E1 10.706,E2 301.0258} C_DIS
LIN {X -118.3871,Y 67.0355,Z 167,A 151.4456,B 10.8433,C 0.0864,E1 10.7037,E2 299.405} C_DIS
LIN {X -120.85,Y 62.4865,Z 167,A 153.521,B 10.8433,C 0.0942,E1 10.701,E2 297.3447} C_DIS
LIN {X -122.3877,Y 59.4182,Z 167,A 154.9835,B 10.8432,C 0.0977,E1 10.6992,E2 295.8816} C_DIS
LIN {X -123.8623,Y 56.279,Z 167,A 156.4616,B 10.8432,C 0.1013,E1 10.6975,E2 294.4031} C_DIS
LIN {X -125.2307,Y 53.1645,Z 167,A 158.0246,B 10.8432,C 0.1025,E1 10.6958,E2 292.8257} C_DIS
LIN {X -126.5148,Y 50.0321,Z 167,A 159.3352,B 10.8431,C 0.1088,E1 10.6944,E2 291.5308} C_DIS
LIN {X -127.7136,Y 46.8875,Z 167,A 160.7708,B 10.8431,C 0.1123,E1 10.693,E2 290.0946} C_DIS
LIN {X -128.8144,Y 43.7735,Z 167,A 162.2148,B 10.8431,C 0.1152,E1 10.6917,E2 288.6457} C_DIS
LIN {X -129.8619,Y 40.5597,Z 167,A 163.7614,B 10.843,C 0.1167,E1 10.6904,E2 287.0856} C_DIS
LIN {X -130.7972,Y 37.4349,Z 167,A 165.0281,B 10.843,C 0.1228,E1 10.6894,E2 285.8334} C_DIS
LIN {X -131.6642,Y 34.261,Z 167,A 166.4486,B 10.8429,C 0.126,E1 10.6884,E2 284.4103} C_DIS
LIN {X -132.4493,Y 31.0879,Z 167,A 167.8879,B 10.8429,C 0.1287,E1 10.6874,E2 282.9648} C_DIS
LIN {X -133.2698,Y 27.3468,Z 167,A 169.4535,B 10.8428,C 0.1343,E1 10.6865,E2 281.4067} C_DIS
LIN {X -133.8506,Y 24.3475,Z 167,A 170.7275,B 10.8428,C 0.1383,E1 10.6859,E2 280.1356} C_DIS
LIN {X -134.3228,Y 21.6025,Z 167,A 171.9472,B 10.8428,C 0.1408,E1 10.6853,E2 278.9116} C_DIS
LIN {X -134.7965,Y 18.4146,Z 167,A 173.3206,B 10.8427,C 0.1444,E1 10.6848,E2 277.5377} C_DIS
LIN {X -135.2459,Y 14.7396,Z 167,A 174.6993,B 10.8425,C 0.1525,E1 10.6843,E2 276.1827} C_DIS
LIN {X -135.4985,Y 12.2246,Z 167,A 175.994,B 10.8425,C 0.1511,E1 10.684,E2 274.8609} C_DIS
LIN {X -135.7447,Y 9.0884,Z 167,A 177.2999,B 10.8425,C 0.1553,E1 10.6837,E2 273.5588} C_DIS
LIN {X -135.9342,Y 5.5362,Z 167,A 178.8586,B 10.8425,C 0.1585,E1 10.6835,E2 271.9942} C_DIS
LIN {X -136.0251,Y 2.4291,Z 167,A -179.8594,B 10.8425,C 0.1629,E1 10.6835,E2 270.7168} C_DIS
LIN {X -136.0397,Y -1.5515,Z 167,A -178.0955,B 10.8424,C 0.1661,E1 10.6835,E2 268.9439} C_DIS
LIN {X -135.9731,Y -4.5393,Z 167,A -176.8442,B 10.8423,C 0.1699,E1 10.6835,E2 267.6949} C_DIS
LIN {X -135.8127,Y -7.9833,Z 167,A -175.3223,B 10.8423,C 0.1727,E1 10.6838,E2 266.1657} C_DIS
LIN {X -135.5683,Y -11.3985,Z 167,A -173.8871,B 10.8422,C 0.1771,E1 10.6841,E2 264.7327} C_DIS
LIN {X -135.2466,Y -14.7325,Z 167,A -172.4834,B 10.8422,C 0.1813,E1 10.6845,E2 263.3312} C_DIS
LIN {X -134.7904,Y -18.4612,Z 167,A -170.8572,B 10.842,C 0.185,E1 10.6851,E2 261.7012} C_DIS
Enddeposition()
END
